LIN {X 65.903,Y 100.037,Z 70.570,A 180.000,B 0.000,C 180.000} C_DIS
LIN {X 65.874,Y 99.882,Z 70.566,A 180.000,B 0.000,C 180.000} C_DIS
LIN {X 65.837,Y 99.729,Z 70.562,A 180.000,B 0.000,C 180.000} C_DIS
LIN {X 65.796,Y 99.577,Z 70.559,A 180.000,B 0.000,C 180.000} C_DIS
LIN {X 65.755,Y 99.425,Z 70.556,A 180.000,B 0.000,C 180.000} C_DIS
LIN {X 65.713,Y 99.273,Z 70.552,A 180.000,B 0.000,C 180.000} C_DIS
LIN {X 65.665,Y 99.123,Z 70.549,A 180.000,B 0.000,C 180.000} C_DIS
LIN {X 65.611,Y 98.975,Z 70.546,A 180.000,B 0.000,C 180.000} C_DIS
LIN {X 65.556,Y 98.827,Z 70.543,A 180.000,B 0.000,C 180.000} C_DIS
LIN {X 65.501,Y 98.679,Z 70.540,A 180.000,B 0.000,C 180.000} C_DIS
LIN {X 65.443,Y 98.533,Z 70.537,A 180.000,B 0.000,C 180.000} C_DIS
LIN {X 65.376,Y 98.391,Z 70.534,A 180.000,B 0.000,C 180.000} C_DIS
LIN {X 65.308,Y 98.248,Z 70.532,A 180.000,B 0.000,C 180.000} C_DIS
LIN {X 65.241,Y 98.106,Z 70.529,A 180.000,B 0.000,C 180.000} C_DIS
LIN {X 65.171,Y 97.965,Z 70.527,A 180.000,B 0.000,C 180.000} C_DIS
LIN {X 65.014,Y 97.692,Z 70.522,A 180.000,B 0.000,C 180.000} C_DIS
LIN {X 64.853,Y 97.421,Z 70.518,A 180.000,B 0.000,C 180.000} C_DIS
LIN {X 64.674,Y 97.162,Z 70.514,A 180.000,B 0.000,C 180.000} C_DIS
LIN {X 64.491,Y 96.906,Z 70.511,A 180.000,B 0.000,C 180.000} C_DIS
LIN {X 64.291,Y 96.662,Z 70.508,A 180.000,B 0.000,C 180.000} C_DIS
LIN {X 64.086,Y 96.423,Z 70.505,A 180.000,B 0.000,C 180.000} C_DIS
LIN {X 63.980,Y 96.307,Z 70.504,A 180.000,B 0.000,C 180.000} C_DIS
LIN {X 63.868,Y 96.196,Z 70.503,A 180.000,B 0.000,C 180.000} C_DIS
LIN {X 63.643,Y 95.976,Z 70.502,A 180.000,B 0.000,C 180.000} C_DIS
LIN {X 63.528,Y 95.868,Z 70.501,A 180.000,B 0.000,C 180.000} C_DIS
LIN {X 63.407,Y 95.766,Z 70.501,A 180.000,B 0.000,C 180.000} C_DIS
LIN {X 63.164,Y 95.567,Z 70.500,A 180.000,B 0.000,C 180.000} C_DIS
LIN {X 62.980,Y 95.424,Z 70.500,A 180.000,B 0.000,C 180.000} C_DIS
; Cutting Move Starts
LIN {X 62.930,Y 95.388,Z 70.500,A 180.000,B 0.000,C 180.000} C_DIS
LIN {X 62.573,Y 95.145,Z 70.500,A 180.000,B 0.000,C 180.000} C_DIS
LIN {X 62.518,Y 95.109,Z 70.500,A 180.000,B 0.000,C 180.000} C_DIS
LIN {X 62.394,Y 95.033,Z 70.500,A 180.000,B 0.000,C 180.000} C_DIS
LIN {X 62.210,Y 94.930,Z 70.500,A 180.000,B 0.000,C 180.000} C_DIS
LIN {X 62.036,Y 94.833,Z 70.500,A 180.000,B 0.000,C 180.000} C_DIS
LIN {X 61.885,Y 94.751,Z 70.500,A 180.000,B 0.000,C 180.000} C_DIS
LIN {X 61.858,Y 94.738,Z 70.500,A 180.000,B 0.000,C 180.000} C_DIS
LIN {X 61.679,Y 94.656,Z 70.500,A 180.000,B 0.000,C 180.000} C_DIS
LIN {X 61.491,Y 94.573,Z 70.500,A 180.000,B 0.000,C 180.000} C_DIS
LIN {X 61.321,Y 94.497,Z 70.500,A 180.000,B 0.000,C 180.000} C_DIS
LIN {X 61.143,Y 94.430,Z 70.500,A 180.000,B 0.000,C 180.000} C_DIS
LIN {X 60.785,Y 94.307,Z 70.500,A 180.000,B 0.000,C 180.000} C_DIS
LIN {X 60.606,Y 94.250,Z 70.500,A 180.000,B 0.000,C 180.000} C_DIS
LIN {X 60.470,Y 94.215,Z 70.500,A 180.000,B 0.000,C 180.000} C_DIS
LIN {X 60.249,Y 94.160,Z 70.500,A 180.000,B 0.000,C 180.000} C_DIS
LIN {X 60.070,Y 94.116,Z 70.500,A 180.000,B 0.000,C 180.000} C_DIS
LIN {X 59.891,Y 94.081,Z 70.500,A 180.000,B 0.000,C 180.000} C_DIS
LIN {X 59.534,Y 94.025,Z 70.500,A 180.000,B 0.000,C 180.000} C_DIS
LIN {X 59.355,Y 93.999,Z 70.500,A 180.000,B 0.000,C 180.000} C_DIS
LIN {X 59.176,Y 93.983,Z 70.500,A 180.000,B 0.000,C 180.000} C_DIS
LIN {X 58.819,Y 93.959,Z 70.500,A 180.000,B 0.000,C 180.000} C_DIS
LIN {X 58.640,Y 93.951,Z 70.500,A 180.000,B 0.000,C 180.000} C_DIS
LIN {X 58.461,Y 93.954,Z 70.500,A 180.000,B 0.000,C 180.000} C_DIS
LIN {X 58.103,Y 93.962,Z 70.500,A 180.000,B 0.000,C 180.000} C_DIS
LIN {X 57.925,Y 93.973,Z 70.500,A 180.000,B 0.000,C 180.000} C_DIS
LIN {X 57.746,Y 93.992,Z 70.500,A 180.000,B 0.000,C 180.000} C_DIS
LIN {X 57.567,Y 94.012,Z 70.500,A 180.000,B 0.000,C 180.000} C_DIS
LIN {X 57.388,Y 94.033,Z 70.500,A 180.000,B 0.000,C 180.000} C_DIS
LIN {X 57.363,Y 94.036,Z 70.500,A 180.000,B 0.000,C 180.000} C_DIS
LIN {X 57.210,Y 94.063,Z 70.500,A 180.000,B 0.000,C 180.000} C_DIS
LIN {X 56.852,Y 94.135,Z 70.500,A 180.000,B 0.000,C 180.000} C_DIS
LIN {X 56.673,Y 94.174,Z 70.500,A 180.000,B 0.000,C 180.000} C_DIS
LIN {X 56.528,Y 94.215,Z 70.500,A 180.000,B 0.000,C 180.000} C_DIS
LIN {X 56.316,Y 94.278,Z 70.500,A 180.000,B 0.000,C 180.000} C_DIS
LIN {X 56.137,Y 94.331,Z 70.500,A 180.000,B 0.000,C 180.000} C_DIS
LIN {X 55.958,Y 94.392,Z 70.500,A 180.000,B 0.000,C 180.000} C_DIS
LIN {X 55.953,Y 94.394,Z 70.500,A 180.000,B 0.000,C 180.000} C_DIS
LIN {X 55.779,Y 94.462,Z 70.500,A 180.000,B 0.000,C 180.000} C_DIS
LIN {X 55.601,Y 94.533,Z 70.500,A 180.000,B 0.000,C 180.000} C_DIS
LIN {X 55.501,Y 94.573,Z 70.500,A 180.000,B 0.000,C 180.000} C_DIS
LIN {X 55.422,Y 94.606,Z 70.500,A 180.000,B 0.000,C 180.000} C_DIS
LIN {X 55.243,Y 94.693,Z 70.500,A 180.000,B 0.000,C 180.000} C_DIS
LIN {X 55.064,Y 94.782,Z 70.500,A 180.000,B 0.000,C 180.000} C_DIS
LIN {X 54.886,Y 94.872,Z 70.500,A 180.000,B 0.000,C 180.000} C_DIS
LIN {X 54.781,Y 94.930,Z 70.500,A 180.000,B 0.000,C 180.000} C_DIS
LIN {X 54.707,Y 94.975,Z 70.500,A 180.000,B 0.000,C 180.000} C_DIS
LIN {X 54.349,Y 95.195,Z 70.500,A 180.000,B 0.000,C 180.000} C_DIS
LIN {X 54.210,Y 95.288,Z 70.500,A 180.000,B 0.000,C 180.000} C_DIS
LIN {X 54.171,Y 95.316,Z 70.500,A 180.000,B 0.000,C 180.000} C_DIS
LIN {X 53.970,Y 95.466,Z 70.500,A 180.000,B 0.000,C 180.000} C_DIS
LIN {X 53.813,Y 95.583,Z 70.500,A 180.000,B 0.000,C 180.000} C_DIS
LIN {X 53.733,Y 95.645,Z 70.500,A 180.000,B 0.000,C 180.000} C_DIS
LIN {X 53.634,Y 95.729,Z 70.500,A 180.000,B 0.000,C 180.000} C_DIS
LIN {X 53.445,Y 95.899,Z 70.500,A 180.000,B 0.000,C 180.000} C_DIS
LIN {X 53.329,Y 96.003,Z 70.500,A 180.000,B 0.000,C 180.000} C_DIS
LIN {X 53.277,Y 96.050,Z 70.500,A 180.000,B 0.000,C 180.000} C_DIS
LIN {X 53.144,Y 96.181,Z 70.500,A 180.000,B 0.000,C 180.000} C_DIS
LIN {X 52.919,Y 96.421,Z 70.500,A 180.000,B 0.000,C 180.000} C_DIS
LIN {X 52.810,Y 96.539,Z 70.500,A 180.000,B 0.000,C 180.000} C_DIS
LIN {X 52.740,Y 96.619,Z 70.500,A 180.000,B 0.000,C 180.000} C_DIS
LIN {X 52.662,Y 96.718,Z 70.500,A 180.000,B 0.000,C 180.000} C_DIS
LIN {X 52.522,Y 96.897,Z 70.500,A 180.000,B 0.000,C 180.000} C_DIS
LIN {X 52.383,Y 97.075,Z 70.500,A 180.000,B 0.000,C 180.000} C_DIS
LIN {X 52.261,Y 97.254,Z 70.500,A 180.000,B 0.000,C 180.000} C_DIS
LIN {X 52.145,Y 97.433,Z 70.500,A 180.000,B 0.000,C 180.000} C_DIS
LIN {X 52.029,Y 97.612,Z 70.500,A 180.000,B 0.000,C 180.000} C_DIS
LIN {X 52.025,Y 97.618,Z 70.500,A 180.000,B 0.000,C 180.000} C_DIS
LIN {X 51.927,Y 97.790,Z 70.500,A 180.000,B 0.000,C 180.000} C_DIS
LIN {X 51.737,Y 98.148,Z 70.500,A 180.000,B 0.000,C 180.000} C_DIS
LIN {X 51.668,Y 98.287,Z 70.500,A 180.000,B 0.000,C 180.000} C_DIS
LIN {X 51.650,Y 98.327,Z 70.500,A 180.000,B 0.000,C 180.000} C_DIS
LIN {X 51.574,Y 98.505,Z 70.500,A 180.000,B 0.000,C 180.000} C_DIS
LIN {X 51.489,Y 98.708,Z 70.500,A 180.000,B 0.000,C 180.000} C_DIS
LIN {X 51.426,Y 98.863,Z 70.500,A 180.000,B 0.000,C 180.000} C_DIS
LIN {X 51.365,Y 99.042,Z 70.500,A 180.000,B 0.000,C 180.000} C_DIS
LIN {X 51.250,Y 99.399,Z 70.500,A 180.000,B 0.000,C 180.000} C_DIS
LIN {X 51.199,Y 99.578,Z 70.500,A 180.000,B 0.000,C 180.000} C_DIS
LIN {X 51.159,Y 99.757,Z 70.500,A 180.000,B 0.000,C 180.000} C_DIS
LIN {X 51.118,Y 99.936,Z 70.500,A 180.000,B 0.000,C 180.000} C_DIS
LIN {X 51.079,Y 100.114,Z 70.500,A 180.000,B 0.000,C 180.000} C_DIS
LIN {X 51.049,Y 100.293,Z 70.500,A 180.000,B 0.000,C 180.000} C_DIS
LIN {X 51.001,Y 100.651,Z 70.500,A 180.000,B 0.000,C 180.000} C_DIS
LIN {X 50.980,Y 100.829,Z 70.500,A 180.000,B 0.000,C 180.000} C_DIS
LIN {X 50.969,Y 101.008,Z 70.500,A 180.000,B 0.000,C 180.000} C_DIS
LIN {X 50.953,Y 101.385,Z 70.500,A 180.000,B 0.000,C 180.000} C_DIS
LIN {X 50.950,Y 101.545,Z 70.500,A 180.000,B 0.000,C 180.000} C_DIS
LIN {X 50.953,Y 101.615,Z 70.500,A 180.000,B 0.000,C 180.000} C_DIS
LIN {X 50.965,Y 101.902,Z 70.500,A 180.000,B 0.000,C 180.000} C_DIS
LIN {X 50.973,Y 102.081,Z 70.500,A 180.000,B 0.000,C 180.000} C_DIS
LIN {X 50.989,Y 102.260,Z 70.500,A 180.000,B 0.000,C 180.000} C_DIS
LIN {X 51.013,Y 102.438,Z 70.500,A 180.000,B 0.000,C 180.000} C_DIS
LIN {X 51.037,Y 102.617,Z 70.500,A 180.000,B 0.000,C 180.000} C_DIS
LIN {X 51.062,Y 102.796,Z 70.500,A 180.000,B 0.000,C 180.000} C_DIS
LIN {X 51.098,Y 102.975,Z 70.500,A 180.000,B 0.000,C 180.000} C_DIS
LIN {X 51.179,Y 103.332,Z 70.500,A 180.000,B 0.000,C 180.000} C_DIS
LIN {X 51.223,Y 103.511,Z 70.500,A 180.000,B 0.000,C 180.000} C_DIS
LIN {X 51.279,Y 103.690,Z 70.500,A 180.000,B 0.000,C 180.000} C_DIS
LIN {X 51.336,Y 103.869,Z 70.500,A 180.000,B 0.000,C 180.000} C_DIS
LIN {X 51.393,Y 104.047,Z 70.500,A 180.000,B 0.000,C 180.000} C_DIS
LIN {X 51.461,Y 104.226,Z 70.500,A 180.000,B 0.000,C 180.000} C_DIS
LIN {X 51.612,Y 104.584,Z 70.500,A 180.000,B 0.000,C 180.000} C_DIS
LIN {X 51.668,Y 104.713,Z 70.500,A 180.000,B 0.000,C 180.000} C_DIS
LIN {X 51.691,Y 104.762,Z 70.500,A 180.000,B 0.000,C 180.000} C_DIS
LIN {X 51.785,Y 104.941,Z 70.500,A 180.000,B 0.000,C 180.000} C_DIS
LIN {X 51.879,Y 105.120,Z 70.500,A 180.000,B 0.000,C 180.000} C_DIS
LIN {X 51.975,Y 105.299,Z 70.500,A 180.000,B 0.000,C 180.000} C_DIS
LIN {X 52.025,Y 105.382,Z 70.500,A 180.000,B 0.000,C 180.000} C_DIS
LIN {X 52.087,Y 105.477,Z 70.500,A 180.000,B 0.000,C 180.000} C_DIS
LIN {X 52.204,Y 105.658,Z 70.500,A 180.000,B 0.000,C 180.000} C_DIS
LIN {X 52.319,Y 105.835,Z 70.500,A 180.000,B 0.000,C 180.000} C_DIS
LIN {X 52.383,Y 105.925,Z 70.500,A 180.000,B 0.000,C 180.000} C_DIS
LIN {X 52.452,Y 106.014,Z 70.500,A 180.000,B 0.000,C 180.000} C_DIS
LIN {X 52.591,Y 106.193,Z 70.500,A 180.000,B 0.000,C 180.000} C_DIS
LIN {X 52.732,Y 106.371,Z 70.500,A 180.000,B 0.000,C 180.000} C_DIS
LIN {X 52.740,Y 106.381,Z 70.500,A 180.000,B 0.000,C 180.000} C_DIS
LIN {X 52.892,Y 106.550,Z 70.500,A 180.000,B 0.000,C 180.000} C_DIS
LIN {X 53.098,Y 106.770,Z 70.500,A 180.000,B 0.000,C 180.000} C_DIS
LIN {X 53.231,Y 106.908,Z 70.500,A 180.000,B 0.000,C 180.000} C_DIS
LIN {X 53.277,Y 106.950,Z 70.500,A 180.000,B 0.000,C 180.000} C_DIS
LIN {X 53.428,Y 107.086,Z 70.500,A 180.000,B 0.000,C 180.000} C_DIS
LIN {X 53.634,Y 107.271,Z 70.500,A 180.000,B 0.000,C 180.000} C_DIS
LIN {X 53.724,Y 107.347,Z 70.500,A 180.000,B 0.000,C 180.000} C_DIS
LIN {X 53.813,Y 107.417,Z 70.500,A 180.000,B 0.000,C 180.000} C_DIS
LIN {X 54.089,Y 107.623,Z 70.500,A 180.000,B 0.000,C 180.000} C_DIS
LIN {X 54.171,Y 107.684,Z 70.500,A 180.000,B 0.000,C 180.000} C_DIS
LIN {X 54.344,Y 107.802,Z 70.500,A 180.000,B 0.000,C 180.000} C_DIS
LIN {X 54.707,Y 108.025,Z 70.500,A 180.000,B 0.000,C 180.000} C_DIS
LIN {X 54.886,Y 108.128,Z 70.500,A 180.000,B 0.000,C 180.000} C_DIS
LIN {X 54.947,Y 108.159,Z 70.500,A 180.000,B 0.000,C 180.000} C_DIS
LIN {X 55.304,Y 108.338,Z 70.500,A 180.000,B 0.000,C 180.000} C_DIS
LIN {X 55.422,Y 108.394,Z 70.500,A 180.000,B 0.000,C 180.000} C_DIS
LIN {X 55.601,Y 108.467,Z 70.500,A 180.000,B 0.000,C 180.000} C_DIS
LIN {X 55.779,Y 108.538,Z 70.500,A 180.000,B 0.000,C 180.000} C_DIS
LIN {X 55.958,Y 108.608,Z 70.500,A 180.000,B 0.000,C 180.000} C_DIS
LIN {X 56.137,Y 108.669,Z 70.500,A 180.000,B 0.000,C 180.000} C_DIS
LIN {X 56.225,Y 108.695,Z 70.500,A 180.000,B 0.000,C 180.000} C_DIS
LIN {X 56.495,Y 108.775,Z 70.500,A 180.000,B 0.000,C 180.000} C_DIS
LIN {X 56.673,Y 108.826,Z 70.500,A 180.000,B 0.000,C 180.000} C_DIS
LIN {X 56.852,Y 108.865,Z 70.500,A 180.000,B 0.000,C 180.000} C_DIS
LIN {X 57.210,Y 108.937,Z 70.500,A 180.000,B 0.000,C 180.000} C_DIS
LIN {X 57.388,Y 108.967,Z 70.500,A 180.000,B 0.000,C 180.000} C_DIS
LIN {X 57.567,Y 108.988,Z 70.500,A 180.000,B 0.000,C 180.000} C_DIS
LIN {X 57.746,Y 109.008,Z 70.500,A 180.000,B 0.000,C 180.000} C_DIS
LIN {X 57.925,Y 109.027,Z 70.500,A 180.000,B 0.000,C 180.000} C_DIS
LIN {X 58.103,Y 109.038,Z 70.500,A 180.000,B 0.000,C 180.000} C_DIS
LIN {X 58.461,Y 109.046,Z 70.500,A 180.000,B 0.000,C 180.000} C_DIS
LIN {X 58.640,Y 109.049,Z 70.500,A 180.000,B 0.000,C 180.000} C_DIS
LIN {X 58.819,Y 109.041,Z 70.500,A 180.000,B 0.000,C 180.000} C_DIS
LIN {X 59.176,Y 109.017,Z 70.500,A 180.000,B 0.000,C 180.000} C_DIS
LIN {X 59.355,Y 109.001,Z 70.500,A 180.000,B 0.000,C 180.000} C_DIS
LIN {X 59.534,Y 108.975,Z 70.500,A 180.000,B 0.000,C 180.000} C_DIS
LIN {X 59.891,Y 108.919,Z 70.500,A 180.000,B 0.000,C 180.000} C_DIS
LIN {X 60.070,Y 108.884,Z 70.500,A 180.000,B 0.000,C 180.000} C_DIS
LIN {X 60.111,Y 108.874,Z 70.500,A 180.000,B 0.000,C 180.000} C_DIS
LIN {X 60.427,Y 108.796,Z 70.500,A 180.000,B 0.000,C 180.000} C_DIS
LIN {X 60.606,Y 108.750,Z 70.500,A 180.000,B 0.000,C 180.000} C_DIS
LIN {X 60.778,Y 108.695,Z 70.500,A 180.000,B 0.000,C 180.000} C_DIS
LIN {X 61.143,Y 108.570,Z 70.500,A 180.000,B 0.000,C 180.000} C_DIS
LIN {X 61.287,Y 108.517,Z 70.500,A 180.000,B 0.000,C 180.000} C_DIS
LIN {X 61.321,Y 108.503,Z 70.500,A 180.000,B 0.000,C 180.000} C_DIS
LIN {X 61.500,Y 108.424,Z 70.500,A 180.000,B 0.000,C 180.000} C_DIS
LIN {X 61.692,Y 108.338,Z 70.500,A 180.000,B 0.000,C 180.000} C_DIS
LIN {X 61.858,Y 108.262,Z 70.500,A 180.000,B 0.000,C 180.000} C_DIS
LIN {X 62.036,Y 108.167,Z 70.500,A 180.000,B 0.000,C 180.000} C_DIS
LIN {X 62.371,Y 107.980,Z 70.500,A 180.000,B 0.000,C 180.000} C_DIS
LIN {X 62.394,Y 107.967,Z 70.500,A 180.000,B 0.000,C 180.000} C_DIS
LIN {X 62.573,Y 107.855,Z 70.500,A 180.000,B 0.000,C 180.000} C_DIS
LIN {X 62.930,Y 107.612,Z 70.500,A 180.000,B 0.000,C 180.000} C_DIS
LIN {X 63.020,Y 107.548,Z 70.500,A 180.000,B 0.000,C 180.000} C_DIS
LIN {X 63.109,Y 107.478,Z 70.500,A 180.000,B 0.000,C 180.000} C_DIS
LIN {X 63.369,Y 107.265,Z 70.500,A 180.000,B 0.000,C 180.000} C_DIS
LIN {X 63.467,Y 107.185,Z 70.500,A 180.000,B 0.000,C 180.000} C_DIS
LIN {X 63.578,Y 107.086,Z 70.500,A 180.000,B 0.000,C 180.000} C_DIS
LIN {X 63.645,Y 107.021,Z 70.500,A 180.000,B 0.000,C 180.000} C_DIS
LIN {X 63.824,Y 106.847,Z 70.500,A 180.000,B 0.000,C 180.000} C_DIS
LIN {X 63.944,Y 106.729,Z 70.500,A 180.000,B 0.000,C 180.000} C_DIS
LIN {X 64.003,Y 106.669,Z 70.500,A 180.000,B 0.000,C 180.000} C_DIS
LIN {X 64.109,Y 106.550,Z 70.500,A 180.000,B 0.000,C 180.000} C_DIS
LIN {X 64.360,Y 106.256,Z 70.500,A 180.000,B 0.000,C 180.000} C_DIS
LIN {X 64.414,Y 106.193,Z 70.500,A 180.000,B 0.000,C 180.000} C_DIS
LIN {X 64.539,Y 106.026,Z 70.500,A 180.000,B 0.000,C 180.000} C_DIS
LIN {X 64.718,Y 105.776,Z 70.500,A 180.000,B 0.000,C 180.000} C_DIS
LIN {X 64.802,Y 105.656,Z 70.500,A 180.000,B 0.000,C 180.000} C_DIS
LIN {X 64.897,Y 105.507,Z 70.500,A 180.000,B 0.000,C 180.000} C_DIS
LIN {X 65.075,Y 105.203,Z 70.500,A 180.000,B 0.000,C 180.000} C_DIS
LIN {X 65.124,Y 105.120,Z 70.500,A 180.000,B 0.000,C 180.000} C_DIS
LIN {X 65.219,Y 104.941,Z 70.500,A 180.000,B 0.000,C 180.000} C_DIS
LIN {X 65.254,Y 104.866,Z 70.500,A 180.000,B 0.000,C 180.000} C_DIS
LIN {X 65.388,Y 104.584,Z 70.500,A 180.000,B 0.000,C 180.000} C_DIS
LIN {X 65.433,Y 104.488,Z 70.500,A 180.000,B 0.000,C 180.000} C_DIS
LIN {X 65.469,Y 104.405,Z 70.500,A 180.000,B 0.000,C 180.000} C_DIS
LIN {X 65.536,Y 104.226,Z 70.500,A 180.000,B 0.000,C 180.000} C_DIS
LIN {X 65.612,Y 104.022,Z 70.500,A 180.000,B 0.000,C 180.000} C_DIS
LIN {X 65.668,Y 103.869,Z 70.500,A 180.000,B 0.000,C 180.000} C_DIS
LIN {X 65.724,Y 103.690,Z 70.500,A 180.000,B 0.000,C 180.000} C_DIS
LIN {X 65.821,Y 103.332,Z 70.500,A 180.000,B 0.000,C 180.000} C_DIS
LIN {X 65.867,Y 103.153,Z 70.500,A 180.000,B 0.000,C 180.000} C_DIS
LIN {X 65.901,Y 102.975,Z 70.500,A 180.000,B 0.000,C 180.000} C_DIS
LIN {X 65.965,Y 102.617,Z 70.500,A 180.000,B 0.000,C 180.000} C_DIS
LIN {X 65.969,Y 102.592,Z 70.500,A 180.000,B 0.000,C 180.000} C_DIS
LIN {X 65.991,Y 102.438,Z 70.500,A 180.000,B 0.000,C 180.000} C_DIS
LIN {X 66.007,Y 102.260,Z 70.500,A 180.000,B 0.000,C 180.000} C_DIS
LIN {X 66.023,Y 102.081,Z 70.500,A 180.000,B 0.000,C 180.000} C_DIS
LIN {X 66.039,Y 101.902,Z 70.500,A 180.000,B 0.000,C 180.000} C_DIS
LIN {X 66.045,Y 101.723,Z 70.500,A 180.000,B 0.000,C 180.000} C_DIS
LIN {X 66.045,Y 101.366,Z 70.500,A 180.000,B 0.000,C 180.000} C_DIS
LIN {X 66.043,Y 101.187,Z 70.500,A 180.000,B 0.000,C 180.000} C_DIS
LIN {X 66.031,Y 101.008,Z 70.500,A 180.000,B 0.000,C 180.000} C_DIS
LIN {X 65.999,Y 100.651,Z 70.500,A 180.000,B 0.000,C 180.000} C_DIS
LIN {X 65.980,Y 100.472,Z 70.500,A 180.000,B 0.000,C 180.000} C_DIS
LIN {X 65.969,Y 100.408,Z 70.500,A 180.000,B 0.000,C 180.000} C_DIS
LIN {X 65.949,Y 100.293,Z 70.500,A 180.000,B 0.000,C 180.000} C_DIS
LIN {X 65.917,Y 100.114,Z 70.500,A 180.000,B 0.000,C 180.000} C_DIS
LIN {X 65.885,Y 99.936,Z 70.500,A 180.000,B 0.000,C 180.000} C_DIS
LIN {X 65.845,Y 99.757,Z 70.500,A 180.000,B 0.000,C 180.000} C_DIS
LIN {X 65.796,Y 99.578,Z 70.500,A 180.000,B 0.000,C 180.000} C_DIS
LIN {X 65.748,Y 99.399,Z 70.500,A 180.000,B 0.000,C 180.000} C_DIS
LIN {X 65.698,Y 99.221,Z 70.500,A 180.000,B 0.000,C 180.000} C_DIS
LIN {X 65.635,Y 99.042,Z 70.500,A 180.000,B 0.000,C 180.000} C_DIS
LIN {X 65.503,Y 98.684,Z 70.500,A 180.000,B 0.000,C 180.000} C_DIS
LIN {X 65.433,Y 98.512,Z 70.500,A 180.000,B 0.000,C 180.000} C_DIS
LIN {X 65.430,Y 98.505,Z 70.500,A 180.000,B 0.000,C 180.000} C_DIS
LIN {X 65.346,Y 98.327,Z 70.500,A 180.000,B 0.000,C 180.000} C_DIS
LIN {X 65.254,Y 98.134,Z 70.500,A 180.000,B 0.000,C 180.000} C_DIS
LIN {X 65.174,Y 97.969,Z 70.500,A 180.000,B 0.000,C 180.000} C_DIS
LIN {X 65.075,Y 97.797,Z 70.500,A 180.000,B 0.000,C 180.000} C_DIS
LIN {X 64.897,Y 97.493,Z 70.500,A 180.000,B 0.000,C 180.000} C_DIS
LIN {X 64.861,Y 97.433,Z 70.500,A 180.000,B 0.000,C 180.000} C_DIS
LIN {X 64.739,Y 97.254,Z 70.500,A 180.000,B 0.000,C 180.000} C_DIS
LIN {X 64.539,Y 96.974,Z 70.500,A 180.000,B 0.000,C 180.000} C_DIS
LIN {X 64.484,Y 96.897,Z 70.500,A 180.000,B 0.000,C 180.000} C_DIS
LIN {X 64.360,Y 96.744,Z 70.500,A 180.000,B 0.000,C 180.000} C_DIS
LIN {X 64.182,Y 96.535,Z 70.500,A 180.000,B 0.000,C 180.000} C_DIS
LIN {X 64.030,Y 96.360,Z 70.500,A 180.000,B 0.000,C 180.000} C_DIS
LIN {X 64.003,Y 96.331,Z 70.500,A 180.000,B 0.000,C 180.000} C_DIS
LIN {X 63.853,Y 96.181,Z 70.500,A 180.000,B 0.000,C 180.000} C_DIS
LIN {X 63.645,Y 95.979,Z 70.500,A 180.000,B 0.000,C 180.000} C_DIS
LIN {X 63.477,Y 95.824,Z 70.500,A 180.000,B 0.000,C 180.000} C_DIS
LIN {X 63.467,Y 95.815,Z 70.500,A 180.000,B 0.000,C 180.000} C_DIS
LIN {X 63.288,Y 95.669,Z 70.500,A 180.000,B 0.000,C 180.000} C_DIS
LIN {X 63.109,Y 95.522,Z 70.500,A 180.000,B 0.000,C 180.000} C_DIS
LIN {X 63.038,Y 95.466,Z 70.500,A 180.000,B 0.000,C 180.000} C_DIS
LIN {X 62.980,Y 95.424,Z 70.500,A 180.000,B 0.000,C 180.000} C_DIS
; Link Move Starts
LIN {X 62.722,Y 95.246,Z 70.499,A 180.000,B 0.000,C 180.000} C_DIS
LIN {X 62.461,Y 95.072,Z 70.496,A 180.000,B 0.000,C 180.000} C_DIS
LIN {X 62.188,Y 94.918,Z 70.492,A 180.000,B 0.000,C 180.000} C_DIS
LIN {X 62.051,Y 94.841,Z 70.489,A 180.000,B 0.000,C 180.000} C_DIS
LIN {X 61.914,Y 94.766,Z 70.486,A 180.000,B 0.000,C 180.000} C_DIS
LIN {X 61.772,Y 94.698,Z 70.482,A 180.000,B 0.000,C 180.000} C_DIS
LIN {X 61.629,Y 94.634,Z 70.479,A 180.000,B 0.000,C 180.000} C_DIS
LIN {X 61.486,Y 94.570,Z 70.475,A 180.000,B 0.000,C 180.000} C_DIS
LIN {X 61.343,Y 94.506,Z 70.470,A 180.000,B 0.000,C 180.000} C_DIS
LIN {X 61.197,Y 94.449,Z 70.465,A 180.000,B 0.000,C 180.000} C_DIS
LIN {X 61.049,Y 94.398,Z 70.460,A 180.000,B 0.000,C 180.000} C_DIS
LIN {X 60.975,Y 94.372,Z 70.458,A 180.000,B 0.000,C 180.000} C_DIS
LIN {X 60.900,Y 94.347,Z 70.455,A 180.000,B 0.000,C 180.000} C_DIS
LIN {X 60.826,Y 94.321,Z 70.453,A 180.000,B 0.000,C 180.000} C_DIS
LIN {X 60.752,Y 94.296,Z 70.450,A 180.000,B 0.000,C 180.000} C_DIS
LIN {X 60.678,Y 94.271,Z 70.447,A 180.000,B 0.000,C 180.000} C_DIS
LIN {X 60.603,Y 94.249,Z 70.444,A 180.000,B 0.000,C 180.000} C_DIS
LIN {X 60.527,Y 94.229,Z 70.442,A 180.000,B 0.000,C 180.000} C_DIS
LIN {X 60.451,Y 94.210,Z 70.439,A 180.000,B 0.000,C 180.000} C_DIS
LIN {X 60.375,Y 94.191,Z 70.436,A 180.000,B 0.000,C 180.000} C_DIS
LIN {X 60.298,Y 94.172,Z 70.433,A 180.000,B 0.000,C 180.000} C_DIS
LIN {X 60.222,Y 94.153,Z 70.431,A 180.000,B 0.000,C 180.000} C_DIS
LIN {X 60.146,Y 94.135,Z 70.428,A 180.000,B 0.000,C 180.000} C_DIS
LIN {X 60.070,Y 94.116,Z 70.425,A 180.000,B 0.000,C 180.000} C_DIS
LIN {X 59.994,Y 94.099,Z 70.422,A 180.000,B 0.000,C 180.000} C_DIS
LIN {X 59.916,Y 94.085,Z 70.420,A 180.000,B 0.000,C 180.000} C_DIS
LIN {X 59.839,Y 94.073,Z 70.417,A 180.000,B 0.000,C 180.000} C_DIS
LIN {X 59.762,Y 94.060,Z 70.414,A 180.000,B 0.000,C 180.000} C_DIS
LIN {X 59.684,Y 94.048,Z 70.411,A 180.000,B 0.000,C 180.000} C_DIS
LIN {X 59.607,Y 94.036,Z 70.409,A 180.000,B 0.000,C 180.000} C_DIS
LIN {X 59.529,Y 94.024,Z 70.406,A 180.000,B 0.000,C 180.000} C_DIS
LIN {X 59.452,Y 94.012,Z 70.403,A 180.000,B 0.000,C 180.000} C_DIS
LIN {X 59.374,Y 94.001,Z 70.401,A 180.000,B 0.000,C 180.000} C_DIS
LIN {X 59.296,Y 93.992,Z 70.398,A 180.000,B 0.000,C 180.000} C_DIS
LIN {X 59.218,Y 93.986,Z 70.395,A 180.000,B 0.000,C 180.000} C_DIS
LIN {X 59.062,Y 93.976,Z 70.390,A 180.000,B 0.000,C 180.000} C_DIS
LIN {X 58.827,Y 93.960,Z 70.381,A 180.000,B 0.000,C 180.000} C_DIS
LIN {X 58.749,Y 93.955,Z 70.379,A 180.000,B 0.000,C 180.000} C_DIS
LIN {X 58.670,Y 93.952,Z 70.376,A 180.000,B 0.000,C 180.000} C_DIS
LIN {X 58.592,Y 93.951,Z 70.373,A 180.000,B 0.000,C 180.000} C_DIS
LIN {X 58.514,Y 93.953,Z 70.370,A 180.000,B 0.000,C 180.000} C_DIS
LIN {X 58.122,Y 93.961,Z 70.357,A 180.000,B 0.000,C 180.000} C_DIS
LIN {X 58.043,Y 93.964,Z 70.354,A 180.000,B 0.000,C 180.000} C_DIS
LIN {X 57.965,Y 93.969,Z 70.351,A 180.000,B 0.000,C 180.000} C_DIS
LIN {X 57.887,Y 93.977,Z 70.348,A 180.000,B 0.000,C 180.000} C_DIS
LIN {X 57.731,Y 93.994,Z 70.343,A 180.000,B 0.000,C 180.000} C_DIS
LIN {X 57.653,Y 94.003,Z 70.340,A 180.000,B 0.000,C 180.000} C_DIS
LIN {X 57.575,Y 94.011,Z 70.338,A 180.000,B 0.000,C 180.000} C_DIS
LIN {X 57.497,Y 94.020,Z 70.335,A 180.000,B 0.000,C 180.000} C_DIS
LIN {X 57.420,Y 94.029,Z 70.332,A 180.000,B 0.000,C 180.000} C_DIS
LIN {X 57.342,Y 94.039,Z 70.329,A 180.000,B 0.000,C 180.000} C_DIS
LIN {X 57.265,Y 94.052,Z 70.327,A 180.000,B 0.000,C 180.000} C_DIS
LIN {X 57.188,Y 94.068,Z 70.324,A 180.000,B 0.000,C 180.000} C_DIS
LIN {X 57.111,Y 94.083,Z 70.321,A 180.000,B 0.000,C 180.000} C_DIS
LIN {X 57.034,Y 94.099,Z 70.318,A 180.000,B 0.000,C 180.000} C_DIS
LIN {X 56.957,Y 94.114,Z 70.316,A 180.000,B 0.000,C 180.000} C_DIS
LIN {X 56.880,Y 94.130,Z 70.313,A 180.000,B 0.000,C 180.000} C_DIS
LIN {X 56.803,Y 94.145,Z 70.310,A 180.000,B 0.000,C 180.000} C_DIS
LIN {X 56.727,Y 94.162,Z 70.307,A 180.000,B 0.000,C 180.000} C_DIS
LIN {X 56.651,Y 94.180,Z 70.305,A 180.000,B 0.000,C 180.000} C_DIS
LIN {X 56.575,Y 94.201,Z 70.302,A 180.000,B 0.000,C 180.000} C_DIS
LIN {X 56.500,Y 94.223,Z 70.299,A 180.000,B 0.000,C 180.000} C_DIS
LIN {X 56.425,Y 94.246,Z 70.297,A 180.000,B 0.000,C 180.000} C_DIS
LIN {X 56.349,Y 94.268,Z 70.294,A 180.000,B 0.000,C 180.000} C_DIS
LIN {X 56.274,Y 94.290,Z 70.291,A 180.000,B 0.000,C 180.000} C_DIS
LIN {X 56.199,Y 94.312,Z 70.288,A 180.000,B 0.000,C 180.000} C_DIS
LIN {X 56.124,Y 94.335,Z 70.286,A 180.000,B 0.000,C 180.000} C_DIS
LIN {X 55.976,Y 94.385,Z 70.281,A 180.000,B 0.000,C 180.000} C_DIS
LIN {X 55.830,Y 94.442,Z 70.276,A 180.000,B 0.000,C 180.000} C_DIS
LIN {X 55.684,Y 94.500,Z 70.272,A 180.000,B 0.000,C 180.000} C_DIS
LIN {X 55.538,Y 94.558,Z 70.268,A 180.000,B 0.000,C 180.000} C_DIS
LIN {X 55.394,Y 94.619,Z 70.264,A 180.000,B 0.000,C 180.000} C_DIS
LIN {X 55.253,Y 94.688,Z 70.260,A 180.000,B 0.000,C 180.000} C_DIS
LIN {X 55.113,Y 94.758,Z 70.257,A 180.000,B 0.000,C 180.000} C_DIS
LIN {X 54.972,Y 94.828,Z 70.255,A 180.000,B 0.000,C 180.000} C_DIS
LIN {X 54.833,Y 94.900,Z 70.252,A 180.000,B 0.000,C 180.000} C_DIS
LIN {X 54.698,Y 94.980,Z 70.250,A 180.000,B 0.000,C 180.000} C_DIS
LIN {X 54.431,Y 95.145,Z 70.247,A 180.000,B 0.000,C 180.000} C_DIS
LIN {X 54.177,Y 95.312,Z 70.247,A 180.000,B 0.000,C 180.000} C_DIS
; Cutting Move Starts
LIN {X 54.171,Y 95.316,Z 70.247,A 180.000,B 0.000,C 180.000} C_DIS
LIN {X 53.970,Y 95.466,Z 70.247,A 180.000,B 0.000,C 180.000} C_DIS
LIN {X 53.813,Y 95.583,Z 70.247,A 180.000,B 0.000,C 180.000} C_DIS
LIN {X 53.733,Y 95.645,Z 70.247,A 180.000,B 0.000,C 180.000} C_DIS
LIN {X 53.634,Y 95.729,Z 70.247,A 180.000,B 0.000,C 180.000} C_DIS
LIN {X 53.329,Y 96.003,Z 70.247,A 180.000,B 0.000,C 180.000} C_DIS
LIN {X 53.277,Y 96.050,Z 70.247,A 180.000,B 0.000,C 180.000} C_DIS
LIN {X 53.144,Y 96.181,Z 70.247,A 180.000,B 0.000,C 180.000} C_DIS
LIN {X 52.919,Y 96.421,Z 70.247,A 180.000,B 0.000,C 180.000} C_DIS
LIN {X 52.810,Y 96.539,Z 70.247,A 180.000,B 0.000,C 180.000} C_DIS
LIN {X 52.740,Y 96.619,Z 70.247,A 180.000,B 0.000,C 180.000} C_DIS
LIN {X 52.662,Y 96.718,Z 70.247,A 180.000,B 0.000,C 180.000} C_DIS
LIN {X 52.522,Y 96.897,Z 70.247,A 180.000,B 0.000,C 180.000} C_DIS
LIN {X 52.383,Y 97.075,Z 70.247,A 180.000,B 0.000,C 180.000} C_DIS
LIN {X 52.261,Y 97.254,Z 70.247,A 180.000,B 0.000,C 180.000} C_DIS
LIN {X 52.145,Y 97.433,Z 70.247,A 180.000,B 0.000,C 180.000} C_DIS
LIN {X 52.029,Y 97.612,Z 70.247,A 180.000,B 0.000,C 180.000} C_DIS
LIN {X 52.025,Y 97.618,Z 70.247,A 180.000,B 0.000,C 180.000} C_DIS
LIN {X 51.927,Y 97.790,Z 70.247,A 180.000,B 0.000,C 180.000} C_DIS
LIN {X 51.737,Y 98.148,Z 70.247,A 180.000,B 0.000,C 180.000} C_DIS
LIN {X 51.668,Y 98.287,Z 70.247,A 180.000,B 0.000,C 180.000} C_DIS
LIN {X 51.650,Y 98.327,Z 70.247,A 180.000,B 0.000,C 180.000} C_DIS
LIN {X 51.574,Y 98.505,Z 70.247,A 180.000,B 0.000,C 180.000} C_DIS
LIN {X 51.489,Y 98.708,Z 70.247,A 180.000,B 0.000,C 180.000} C_DIS
LIN {X 51.426,Y 98.863,Z 70.247,A 180.000,B 0.000,C 180.000} C_DIS
LIN {X 51.365,Y 99.042,Z 70.247,A 180.000,B 0.000,C 180.000} C_DIS
LIN {X 51.250,Y 99.399,Z 70.247,A 180.000,B 0.000,C 180.000} C_DIS
LIN {X 51.199,Y 99.578,Z 70.247,A 180.000,B 0.000,C 180.000} C_DIS
LIN {X 51.159,Y 99.757,Z 70.247,A 180.000,B 0.000,C 180.000} C_DIS
LIN {X 51.118,Y 99.936,Z 70.247,A 180.000,B 0.000,C 180.000} C_DIS
LIN {X 51.079,Y 100.114,Z 70.247,A 180.000,B 0.000,C 180.000} C_DIS
LIN {X 51.049,Y 100.293,Z 70.247,A 180.000,B 0.000,C 180.000} C_DIS
LIN {X 51.001,Y 100.651,Z 70.247,A 180.000,B 0.000,C 180.000} C_DIS
LIN {X 50.980,Y 100.829,Z 70.247,A 180.000,B 0.000,C 180.000} C_DIS
LIN {X 50.969,Y 101.008,Z 70.247,A 180.000,B 0.000,C 180.000} C_DIS
LIN {X 50.953,Y 101.385,Z 70.247,A 180.000,B 0.000,C 180.000} C_DIS
LIN {X 50.950,Y 101.545,Z 70.247,A 180.000,B 0.000,C 180.000} C_DIS
LIN {X 50.953,Y 101.615,Z 70.247,A 180.000,B 0.000,C 180.000} C_DIS
LIN {X 50.965,Y 101.902,Z 70.247,A 180.000,B 0.000,C 180.000} C_DIS
LIN {X 50.973,Y 102.081,Z 70.247,A 180.000,B 0.000,C 180.000} C_DIS
LIN {X 50.989,Y 102.260,Z 70.247,A 180.000,B 0.000,C 180.000} C_DIS
LIN {X 51.013,Y 102.438,Z 70.247,A 180.000,B 0.000,C 180.000} C_DIS
LIN {X 51.037,Y 102.617,Z 70.247,A 180.000,B 0.000,C 180.000} C_DIS
LIN {X 51.062,Y 102.796,Z 70.247,A 180.000,B 0.000,C 180.000} C_DIS
LIN {X 51.098,Y 102.975,Z 70.247,A 180.000,B 0.000,C 180.000} C_DIS
LIN {X 51.179,Y 103.332,Z 70.247,A 180.000,B 0.000,C 180.000} C_DIS
LIN {X 51.223,Y 103.511,Z 70.247,A 180.000,B 0.000,C 180.000} C_DIS
LIN {X 51.279,Y 103.690,Z 70.247,A 180.000,B 0.000,C 180.000} C_DIS
LIN {X 51.336,Y 103.869,Z 70.247,A 180.000,B 0.000,C 180.000} C_DIS
LIN {X 51.393,Y 104.047,Z 70.247,A 180.000,B 0.000,C 180.000} C_DIS
LIN {X 51.461,Y 104.226,Z 70.247,A 180.000,B 0.000,C 180.000} C_DIS
LIN {X 51.612,Y 104.584,Z 70.247,A 180.000,B 0.000,C 180.000} C_DIS
LIN {X 51.668,Y 104.713,Z 70.247,A 180.000,B 0.000,C 180.000} C_DIS
LIN {X 51.691,Y 104.762,Z 70.247,A 180.000,B 0.000,C 180.000} C_DIS
LIN {X 51.785,Y 104.941,Z 70.247,A 180.000,B 0.000,C 180.000} C_DIS
LIN {X 51.879,Y 105.120,Z 70.247,A 180.000,B 0.000,C 180.000} C_DIS
LIN {X 51.975,Y 105.299,Z 70.247,A 180.000,B 0.000,C 180.000} C_DIS
LIN {X 52.025,Y 105.382,Z 70.247,A 180.000,B 0.000,C 180.000} C_DIS
LIN {X 52.087,Y 105.477,Z 70.247,A 180.000,B 0.000,C 180.000} C_DIS
LIN {X 52.204,Y 105.658,Z 70.247,A 180.000,B 0.000,C 180.000} C_DIS
LIN {X 52.319,Y 105.835,Z 70.247,A 180.000,B 0.000,C 180.000} C_DIS
LIN {X 52.383,Y 105.925,Z 70.247,A 180.000,B 0.000,C 180.000} C_DIS
LIN {X 52.452,Y 106.014,Z 70.247,A 180.000,B 0.000,C 180.000} C_DIS
LIN {X 52.591,Y 106.193,Z 70.247,A 180.000,B 0.000,C 180.000} C_DIS
LIN {X 52.732,Y 106.371,Z 70.247,A 180.000,B 0.000,C 180.000} C_DIS
LIN {X 52.740,Y 106.381,Z 70.247,A 180.000,B 0.000,C 180.000} C_DIS
LIN {X 52.892,Y 106.550,Z 70.247,A 180.000,B 0.000,C 180.000} C_DIS
LIN {X 53.098,Y 106.770,Z 70.247,A 180.000,B 0.000,C 180.000} C_DIS
LIN {X 53.231,Y 106.908,Z 70.247,A 180.000,B 0.000,C 180.000} C_DIS
LIN {X 53.277,Y 106.950,Z 70.247,A 180.000,B 0.000,C 180.000} C_DIS
LIN {X 53.428,Y 107.086,Z 70.247,A 180.000,B 0.000,C 180.000} C_DIS
LIN {X 53.634,Y 107.271,Z 70.247,A 180.000,B 0.000,C 180.000} C_DIS
LIN {X 53.724,Y 107.347,Z 70.247,A 180.000,B 0.000,C 180.000} C_DIS
LIN {X 53.813,Y 107.417,Z 70.247,A 180.000,B 0.000,C 180.000} C_DIS
LIN {X 54.089,Y 107.623,Z 70.247,A 180.000,B 0.000,C 180.000} C_DIS
LIN {X 54.171,Y 107.684,Z 70.247,A 180.000,B 0.000,C 180.000} C_DIS
LIN {X 54.344,Y 107.802,Z 70.247,A 180.000,B 0.000,C 180.000} C_DIS
LIN {X 54.707,Y 108.025,Z 70.247,A 180.000,B 0.000,C 180.000} C_DIS
LIN {X 54.886,Y 108.128,Z 70.247,A 180.000,B 0.000,C 180.000} C_DIS
LIN {X 54.947,Y 108.159,Z 70.247,A 180.000,B 0.000,C 180.000} C_DIS
LIN {X 55.304,Y 108.338,Z 70.247,A 180.000,B 0.000,C 180.000} C_DIS
LIN {X 55.422,Y 108.394,Z 70.247,A 180.000,B 0.000,C 180.000} C_DIS
LIN {X 55.601,Y 108.467,Z 70.247,A 180.000,B 0.000,C 180.000} C_DIS
LIN {X 55.779,Y 108.538,Z 70.247,A 180.000,B 0.000,C 180.000} C_DIS
LIN {X 55.958,Y 108.608,Z 70.247,A 180.000,B 0.000,C 180.000} C_DIS
LIN {X 56.137,Y 108.669,Z 70.247,A 180.000,B 0.000,C 180.000} C_DIS
LIN {X 56.225,Y 108.695,Z 70.247,A 180.000,B 0.000,C 180.000} C_DIS
LIN {X 56.495,Y 108.775,Z 70.247,A 180.000,B 0.000,C 180.000} C_DIS
LIN {X 56.673,Y 108.826,Z 70.247,A 180.000,B 0.000,C 180.000} C_DIS
LIN {X 56.852,Y 108.865,Z 70.247,A 180.000,B 0.000,C 180.000} C_DIS
LIN {X 57.210,Y 108.937,Z 70.247,A 180.000,B 0.000,C 180.000} C_DIS
LIN {X 57.388,Y 108.967,Z 70.247,A 180.000,B 0.000,C 180.000} C_DIS
LIN {X 57.567,Y 108.988,Z 70.247,A 180.000,B 0.000,C 180.000} C_DIS
LIN {X 57.746,Y 109.008,Z 70.247,A 180.000,B 0.000,C 180.000} C_DIS
LIN {X 57.925,Y 109.027,Z 70.247,A 180.000,B 0.000,C 180.000} C_DIS
LIN {X 58.103,Y 109.038,Z 70.247,A 180.000,B 0.000,C 180.000} C_DIS
LIN {X 58.461,Y 109.046,Z 70.247,A 180.000,B 0.000,C 180.000} C_DIS
LIN {X 58.640,Y 109.049,Z 70.247,A 180.000,B 0.000,C 180.000} C_DIS
LIN {X 58.819,Y 109.041,Z 70.247,A 180.000,B 0.000,C 180.000} C_DIS
LIN {X 59.176,Y 109.017,Z 70.247,A 180.000,B 0.000,C 180.000} C_DIS
LIN {X 59.355,Y 109.001,Z 70.247,A 180.000,B 0.000,C 180.000} C_DIS
LIN {X 59.534,Y 108.975,Z 70.247,A 180.000,B 0.000,C 180.000} C_DIS
LIN {X 59.891,Y 108.919,Z 70.247,A 180.000,B 0.000,C 180.000} C_DIS
LIN {X 60.070,Y 108.884,Z 70.247,A 180.000,B 0.000,C 180.000} C_DIS
LIN {X 60.111,Y 108.874,Z 70.247,A 180.000,B 0.000,C 180.000} C_DIS
LIN {X 60.427,Y 108.796,Z 70.247,A 180.000,B 0.000,C 180.000} C_DIS
LIN {X 60.606,Y 108.750,Z 70.247,A 180.000,B 0.000,C 180.000} C_DIS
LIN {X 60.778,Y 108.695,Z 70.247,A 180.000,B 0.000,C 180.000} C_DIS
LIN {X 61.143,Y 108.570,Z 70.247,A 180.000,B 0.000,C 180.000} C_DIS
LIN {X 61.287,Y 108.517,Z 70.247,A 180.000,B 0.000,C 180.000} C_DIS
LIN {X 61.321,Y 108.503,Z 70.247,A 180.000,B 0.000,C 180.000} C_DIS
LIN {X 61.500,Y 108.424,Z 70.247,A 180.000,B 0.000,C 180.000} C_DIS
LIN {X 61.692,Y 108.338,Z 70.247,A 180.000,B 0.000,C 180.000} C_DIS
LIN {X 61.858,Y 108.262,Z 70.247,A 180.000,B 0.000,C 180.000} C_DIS
LIN {X 62.036,Y 108.167,Z 70.247,A 180.000,B 0.000,C 180.000} C_DIS
LIN {X 62.371,Y 107.980,Z 70.247,A 180.000,B 0.000,C 180.000} C_DIS
LIN {X 62.394,Y 107.967,Z 70.247,A 180.000,B 0.000,C 180.000} C_DIS
LIN {X 62.573,Y 107.855,Z 70.247,A 180.000,B 0.000,C 180.000} C_DIS
LIN {X 62.930,Y 107.612,Z 70.247,A 180.000,B 0.000,C 180.000} C_DIS
LIN {X 63.020,Y 107.548,Z 70.247,A 180.000,B 0.000,C 180.000} C_DIS
LIN {X 63.109,Y 107.478,Z 70.247,A 180.000,B 0.000,C 180.000} C_DIS
LIN {X 63.369,Y 107.265,Z 70.247,A 180.000,B 0.000,C 180.000} C_DIS
LIN {X 63.467,Y 107.185,Z 70.247,A 180.000,B 0.000,C 180.000} C_DIS
LIN {X 63.578,Y 107.086,Z 70.247,A 180.000,B 0.000,C 180.000} C_DIS
LIN {X 63.645,Y 107.021,Z 70.247,A 180.000,B 0.000,C 180.000} C_DIS
LIN {X 63.824,Y 106.847,Z 70.247,A 180.000,B 0.000,C 180.000} C_DIS
LIN {X 63.944,Y 106.729,Z 70.247,A 180.000,B 0.000,C 180.000} C_DIS
LIN {X 64.003,Y 106.669,Z 70.247,A 180.000,B 0.000,C 180.000} C_DIS
LIN {X 64.109,Y 106.550,Z 70.247,A 180.000,B 0.000,C 180.000} C_DIS
LIN {X 64.360,Y 106.256,Z 70.247,A 180.000,B 0.000,C 180.000} C_DIS
LIN {X 64.414,Y 106.193,Z 70.247,A 180.000,B 0.000,C 180.000} C_DIS
LIN {X 64.539,Y 106.026,Z 70.247,A 180.000,B 0.000,C 180.000} C_DIS
LIN {X 64.718,Y 105.776,Z 70.247,A 180.000,B 0.000,C 180.000} C_DIS
LIN {X 64.802,Y 105.656,Z 70.247,A 180.000,B 0.000,C 180.000} C_DIS
LIN {X 64.897,Y 105.507,Z 70.247,A 180.000,B 0.000,C 180.000} C_DIS
LIN {X 65.075,Y 105.203,Z 70.247,A 180.000,B 0.000,C 180.000} C_DIS
LIN {X 65.124,Y 105.120,Z 70.247,A 180.000,B 0.000,C 180.000} C_DIS
LIN {X 65.219,Y 104.941,Z 70.247,A 180.000,B 0.000,C 180.000} C_DIS
LIN {X 65.254,Y 104.866,Z 70.247,A 180.000,B 0.000,C 180.000} C_DIS
LIN {X 65.388,Y 104.584,Z 70.247,A 180.000,B 0.000,C 180.000} C_DIS
LIN {X 65.433,Y 104.488,Z 70.247,A 180.000,B 0.000,C 180.000} C_DIS
LIN {X 65.469,Y 104.405,Z 70.247,A 180.000,B 0.000,C 180.000} C_DIS
LIN {X 65.536,Y 104.226,Z 70.247,A 180.000,B 0.000,C 180.000} C_DIS
LIN {X 65.612,Y 104.022,Z 70.247,A 180.000,B 0.000,C 180.000} C_DIS
LIN {X 65.668,Y 103.869,Z 70.247,A 180.000,B 0.000,C 180.000} C_DIS
LIN {X 65.724,Y 103.690,Z 70.247,A 180.000,B 0.000,C 180.000} C_DIS
LIN {X 65.821,Y 103.332,Z 70.247,A 180.000,B 0.000,C 180.000} C_DIS
LIN {X 65.867,Y 103.153,Z 70.247,A 180.000,B 0.000,C 180.000} C_DIS
LIN {X 65.901,Y 102.975,Z 70.247,A 180.000,B 0.000,C 180.000} C_DIS
LIN {X 65.965,Y 102.617,Z 70.247,A 180.000,B 0.000,C 180.000} C_DIS
LIN {X 65.969,Y 102.592,Z 70.247,A 180.000,B 0.000,C 180.000} C_DIS
LIN {X 65.991,Y 102.438,Z 70.247,A 180.000,B 0.000,C 180.000} C_DIS
LIN {X 66.007,Y 102.260,Z 70.247,A 180.000,B 0.000,C 180.000} C_DIS
LIN {X 66.023,Y 102.081,Z 70.247,A 180.000,B 0.000,C 180.000} C_DIS
LIN {X 66.039,Y 101.902,Z 70.247,A 180.000,B 0.000,C 180.000} C_DIS
LIN {X 66.045,Y 101.723,Z 70.247,A 180.000,B 0.000,C 180.000} C_DIS
LIN {X 66.045,Y 101.366,Z 70.247,A 180.000,B 0.000,C 180.000} C_DIS
LIN {X 66.043,Y 101.187,Z 70.247,A 180.000,B 0.000,C 180.000} C_DIS
LIN {X 66.031,Y 101.008,Z 70.247,A 180.000,B 0.000,C 180.000} C_DIS
LIN {X 65.999,Y 100.651,Z 70.247,A 180.000,B 0.000,C 180.000} C_DIS
LIN {X 65.980,Y 100.472,Z 70.247,A 180.000,B 0.000,C 180.000} C_DIS
LIN {X 65.969,Y 100.408,Z 70.247,A 180.000,B 0.000,C 180.000} C_DIS
LIN {X 65.949,Y 100.293,Z 70.247,A 180.000,B 0.000,C 180.000} C_DIS
LIN {X 65.917,Y 100.114,Z 70.247,A 180.000,B 0.000,C 180.000} C_DIS
LIN {X 65.885,Y 99.936,Z 70.247,A 180.000,B 0.000,C 180.000} C_DIS
LIN {X 65.845,Y 99.757,Z 70.247,A 180.000,B 0.000,C 180.000} C_DIS
LIN {X 65.796,Y 99.578,Z 70.247,A 180.000,B 0.000,C 180.000} C_DIS
LIN {X 65.748,Y 99.399,Z 70.247,A 180.000,B 0.000,C 180.000} C_DIS
LIN {X 65.698,Y 99.221,Z 70.247,A 180.000,B 0.000,C 180.000} C_DIS
LIN {X 65.635,Y 99.042,Z 70.247,A 180.000,B 0.000,C 180.000} C_DIS
LIN {X 65.503,Y 98.684,Z 70.247,A 180.000,B 0.000,C 180.000} C_DIS
LIN {X 65.433,Y 98.512,Z 70.247,A 180.000,B 0.000,C 180.000} C_DIS
LIN {X 65.430,Y 98.505,Z 70.247,A 180.000,B 0.000,C 180.000} C_DIS
LIN {X 65.346,Y 98.327,Z 70.247,A 180.000,B 0.000,C 180.000} C_DIS
LIN {X 65.254,Y 98.134,Z 70.247,A 180.000,B 0.000,C 180.000} C_DIS
LIN {X 65.174,Y 97.969,Z 70.247,A 180.000,B 0.000,C 180.000} C_DIS
LIN {X 65.075,Y 97.797,Z 70.247,A 180.000,B 0.000,C 180.000} C_DIS
LIN {X 64.897,Y 97.493,Z 70.247,A 180.000,B 0.000,C 180.000} C_DIS
LIN {X 64.861,Y 97.433,Z 70.247,A 180.000,B 0.000,C 180.000} C_DIS
LIN {X 64.739,Y 97.254,Z 70.247,A 180.000,B 0.000,C 180.000} C_DIS
LIN {X 64.539,Y 96.974,Z 70.247,A 180.000,B 0.000,C 180.000} C_DIS
LIN {X 64.484,Y 96.897,Z 70.247,A 180.000,B 0.000,C 180.000} C_DIS
LIN {X 64.360,Y 96.744,Z 70.247,A 180.000,B 0.000,C 180.000} C_DIS
LIN {X 64.182,Y 96.535,Z 70.247,A 180.000,B 0.000,C 180.000} C_DIS
LIN {X 64.030,Y 96.360,Z 70.247,A 180.000,B 0.000,C 180.000} C_DIS
LIN {X 64.003,Y 96.331,Z 70.247,A 180.000,B 0.000,C 180.000} C_DIS
LIN {X 63.853,Y 96.181,Z 70.247,A 180.000,B 0.000,C 180.000} C_DIS
LIN {X 63.645,Y 95.979,Z 70.247,A 180.000,B 0.000,C 180.000} C_DIS
LIN {X 63.477,Y 95.824,Z 70.247,A 180.000,B 0.000,C 180.000} C_DIS
LIN {X 63.467,Y 95.815,Z 70.247,A 180.000,B 0.000,C 180.000} C_DIS
LIN {X 63.288,Y 95.669,Z 70.247,A 180.000,B 0.000,C 180.000} C_DIS
LIN {X 63.109,Y 95.522,Z 70.247,A 180.000,B 0.000,C 180.000} C_DIS
LIN {X 63.038,Y 95.466,Z 70.247,A 180.000,B 0.000,C 180.000} C_DIS
LIN {X 62.980,Y 95.424,Z 70.247,A 180.000,B 0.000,C 180.000} C_DIS
LIN {X 62.930,Y 95.388,Z 70.247,A 180.000,B 0.000,C 180.000} C_DIS
LIN {X 62.573,Y 95.145,Z 70.247,A 180.000,B 0.000,C 180.000} C_DIS
LIN {X 62.518,Y 95.109,Z 70.247,A 180.000,B 0.000,C 180.000} C_DIS
LIN {X 62.394,Y 95.033,Z 70.247,A 180.000,B 0.000,C 180.000} C_DIS
LIN {X 62.210,Y 94.930,Z 70.247,A 180.000,B 0.000,C 180.000} C_DIS
LIN {X 62.036,Y 94.833,Z 70.247,A 180.000,B 0.000,C 180.000} C_DIS
LIN {X 61.885,Y 94.751,Z 70.247,A 180.000,B 0.000,C 180.000} C_DIS
LIN {X 61.858,Y 94.738,Z 70.247,A 180.000,B 0.000,C 180.000} C_DIS
LIN {X 61.679,Y 94.656,Z 70.247,A 180.000,B 0.000,C 180.000} C_DIS
LIN {X 61.491,Y 94.573,Z 70.247,A 180.000,B 0.000,C 180.000} C_DIS
LIN {X 61.321,Y 94.497,Z 70.247,A 180.000,B 0.000,C 180.000} C_DIS
LIN {X 61.143,Y 94.430,Z 70.247,A 180.000,B 0.000,C 180.000} C_DIS
LIN {X 60.785,Y 94.307,Z 70.247,A 180.000,B 0.000,C 180.000} C_DIS
LIN {X 60.606,Y 94.250,Z 70.247,A 180.000,B 0.000,C 180.000} C_DIS
LIN {X 60.470,Y 94.215,Z 70.247,A 180.000,B 0.000,C 180.000} C_DIS
LIN {X 60.249,Y 94.160,Z 70.247,A 180.000,B 0.000,C 180.000} C_DIS
LIN {X 60.070,Y 94.116,Z 70.247,A 180.000,B 0.000,C 180.000} C_DIS
LIN {X 59.891,Y 94.081,Z 70.247,A 180.000,B 0.000,C 180.000} C_DIS
LIN {X 59.534,Y 94.025,Z 70.247,A 180.000,B 0.000,C 180.000} C_DIS
LIN {X 59.355,Y 93.999,Z 70.247,A 180.000,B 0.000,C 180.000} C_DIS
LIN {X 59.176,Y 93.983,Z 70.247,A 180.000,B 0.000,C 180.000} C_DIS
LIN {X 58.819,Y 93.959,Z 70.247,A 180.000,B 0.000,C 180.000} C_DIS
LIN {X 58.640,Y 93.951,Z 70.247,A 180.000,B 0.000,C 180.000} C_DIS
LIN {X 58.461,Y 93.954,Z 70.247,A 180.000,B 0.000,C 180.000} C_DIS
LIN {X 58.103,Y 93.962,Z 70.247,A 180.000,B 0.000,C 180.000} C_DIS
LIN {X 57.925,Y 93.973,Z 70.247,A 180.000,B 0.000,C 180.000} C_DIS
LIN {X 57.746,Y 93.992,Z 70.247,A 180.000,B 0.000,C 180.000} C_DIS
LIN {X 57.567,Y 94.012,Z 70.247,A 180.000,B 0.000,C 180.000} C_DIS
LIN {X 57.388,Y 94.033,Z 70.247,A 180.000,B 0.000,C 180.000} C_DIS
LIN {X 57.363,Y 94.036,Z 70.247,A 180.000,B 0.000,C 180.000} C_DIS
LIN {X 57.210,Y 94.063,Z 70.247,A 180.000,B 0.000,C 180.000} C_DIS
LIN {X 56.852,Y 94.135,Z 70.247,A 180.000,B 0.000,C 180.000} C_DIS
LIN {X 56.673,Y 94.174,Z 70.247,A 180.000,B 0.000,C 180.000} C_DIS
LIN {X 56.528,Y 94.215,Z 70.247,A 180.000,B 0.000,C 180.000} C_DIS
LIN {X 56.316,Y 94.278,Z 70.247,A 180.000,B 0.000,C 180.000} C_DIS
LIN {X 56.137,Y 94.331,Z 70.247,A 180.000,B 0.000,C 180.000} C_DIS
LIN {X 55.958,Y 94.392,Z 70.247,A 180.000,B 0.000,C 180.000} C_DIS
LIN {X 55.953,Y 94.394,Z 70.247,A 180.000,B 0.000,C 180.000} C_DIS
LIN {X 55.779,Y 94.462,Z 70.247,A 180.000,B 0.000,C 180.000} C_DIS
LIN {X 55.601,Y 94.533,Z 70.247,A 180.000,B 0.000,C 180.000} C_DIS
LIN {X 55.501,Y 94.573,Z 70.247,A 180.000,B 0.000,C 180.000} C_DIS
LIN {X 55.422,Y 94.606,Z 70.247,A 180.000,B 0.000,C 180.000} C_DIS
LIN {X 55.243,Y 94.693,Z 70.247,A 180.000,B 0.000,C 180.000} C_DIS
LIN {X 55.064,Y 94.782,Z 70.247,A 180.000,B 0.000,C 180.000} C_DIS
LIN {X 54.886,Y 94.872,Z 70.247,A 180.000,B 0.000,C 180.000} C_DIS
LIN {X 54.781,Y 94.930,Z 70.247,A 180.000,B 0.000,C 180.000} C_DIS
LIN {X 54.707,Y 94.975,Z 70.247,A 180.000,B 0.000,C 180.000} C_DIS
LIN {X 54.349,Y 95.195,Z 70.247,A 180.000,B 0.000,C 180.000} C_DIS
LIN {X 54.210,Y 95.288,Z 70.247,A 180.000,B 0.000,C 180.000} C_DIS
LIN {X 54.177,Y 95.312,Z 70.247,A 180.000,B 0.000,C 180.000} C_DIS
; Link Move Starts
LIN {X 53.933,Y 95.494,Z 70.246,A 180.000,B 0.000,C 180.000} C_DIS
LIN {X 53.691,Y 95.680,Z 70.243,A 180.000,B 0.000,C 180.000} C_DIS
LIN {X 53.463,Y 95.883,Z 70.239,A 180.000,B 0.000,C 180.000} C_DIS
LIN {X 53.349,Y 95.985,Z 70.236,A 180.000,B 0.000,C 180.000} C_DIS
LIN {X 53.236,Y 96.087,Z 70.233,A 180.000,B 0.000,C 180.000} C_DIS
LIN {X 53.130,Y 96.196,Z 70.230,A 180.000,B 0.000,C 180.000} C_DIS
LIN {X 53.025,Y 96.308,Z 70.226,A 180.000,B 0.000,C 180.000} C_DIS
LIN {X 52.921,Y 96.419,Z 70.222,A 180.000,B 0.000,C 180.000} C_DIS
LIN {X 52.817,Y 96.531,Z 70.217,A 180.000,B 0.000,C 180.000} C_DIS
LIN {X 52.718,Y 96.647,Z 70.213,A 180.000,B 0.000,C 180.000} C_DIS
LIN {X 52.623,Y 96.767,Z 70.208,A 180.000,B 0.000,C 180.000} C_DIS
LIN {X 52.576,Y 96.827,Z 70.206,A 180.000,B 0.000,C 180.000} C_DIS
LIN {X 52.529,Y 96.887,Z 70.203,A 180.000,B 0.000,C 180.000} C_DIS
LIN {X 52.482,Y 96.947,Z 70.200,A 180.000,B 0.000,C 180.000} C_DIS
LIN {X 52.435,Y 97.007,Z 70.198,A 180.000,B 0.000,C 180.000} C_DIS
LIN {X 52.389,Y 97.067,Z 70.195,A 180.000,B 0.000,C 180.000} C_DIS
LIN {X 52.344,Y 97.129,Z 70.192,A 180.000,B 0.000,C 180.000} C_DIS
LIN {X 52.301,Y 97.192,Z 70.190,A 180.000,B 0.000,C 180.000} C_DIS
LIN {X 52.259,Y 97.256,Z 70.187,A 180.000,B 0.000,C 180.000} C_DIS
LIN {X 52.218,Y 97.320,Z 70.184,A 180.000,B 0.000,C 180.000} C_DIS
LIN {X 52.176,Y 97.384,Z 70.182,A 180.000,B 0.000,C 180.000} C_DIS
LIN {X 52.135,Y 97.448,Z 70.179,A 180.000,B 0.000,C 180.000} C_DIS
LIN {X 52.093,Y 97.512,Z 70.176,A 180.000,B 0.000,C 180.000} C_DIS
LIN {X 52.052,Y 97.576,Z 70.174,A 180.000,B 0.000,C 180.000} C_DIS
LIN {X 52.011,Y 97.641,Z 70.171,A 180.000,B 0.000,C 180.000} C_DIS
LIN {X 51.972,Y 97.707,Z 70.168,A 180.000,B 0.000,C 180.000} C_DIS
LIN {X 51.936,Y 97.773,Z 70.166,A 180.000,B 0.000,C 180.000} C_DIS
LIN {X 51.900,Y 97.841,Z 70.163,A 180.000,B 0.000,C 180.000} C_DIS
LIN {X 51.864,Y 97.908,Z 70.160,A 180.000,B 0.000,C 180.000} C_DIS
LIN {X 51.829,Y 97.976,Z 70.158,A 180.000,B 0.000,C 180.000} C_DIS
LIN {X 51.793,Y 98.043,Z 70.155,A 180.000,B 0.000,C 180.000} C_DIS
LIN {X 51.757,Y 98.111,Z 70.152,A 180.000,B 0.000,C 180.000} C_DIS
LIN {X 51.722,Y 98.178,Z 70.150,A 180.000,B 0.000,C 180.000} C_DIS
LIN {X 51.687,Y 98.246,Z 70.147,A 180.000,B 0.000,C 180.000} C_DIS
LIN {X 51.655,Y 98.315,Z 70.144,A 180.000,B 0.000,C 180.000} C_DIS
LIN {X 51.625,Y 98.385,Z 70.142,A 180.000,B 0.000,C 180.000} C_DIS
LIN {X 51.566,Y 98.526,Z 70.136,A 180.000,B 0.000,C 180.000} C_DIS
LIN {X 51.506,Y 98.667,Z 70.131,A 180.000,B 0.000,C 180.000} C_DIS
LIN {X 51.477,Y 98.737,Z 70.128,A 180.000,B 0.000,C 180.000} C_DIS
LIN {X 51.447,Y 98.807,Z 70.126,A 180.000,B 0.000,C 180.000} C_DIS
LIN {X 51.420,Y 98.878,Z 70.123,A 180.000,B 0.000,C 180.000} C_DIS
LIN {X 51.394,Y 98.950,Z 70.120,A 180.000,B 0.000,C 180.000} C_DIS
LIN {X 51.371,Y 99.023,Z 70.118,A 180.000,B 0.000,C 180.000} C_DIS
LIN {X 51.254,Y 99.386,Z 70.104,A 180.000,B 0.000,C 180.000} C_DIS
LIN {X 51.232,Y 99.459,Z 70.102,A 180.000,B 0.000,C 180.000} C_DIS
LIN {X 51.211,Y 99.533,Z 70.099,A 180.000,B 0.000,C 180.000} C_DIS
LIN {X 51.192,Y 99.607,Z 70.096,A 180.000,B 0.000,C 180.000} C_DIS
LIN {X 51.176,Y 99.681,Z 70.094,A 180.000,B 0.000,C 180.000} C_DIS
LIN {X 51.159,Y 99.755,Z 70.091,A 180.000,B 0.000,C 180.000} C_DIS
LIN {X 51.142,Y 99.830,Z 70.088,A 180.000,B 0.000,C 180.000} C_DIS
LIN {X 51.125,Y 99.904,Z 70.086,A 180.000,B 0.000,C 180.000} C_DIS
LIN {X 51.109,Y 99.979,Z 70.083,A 180.000,B 0.000,C 180.000} C_DIS
LIN {X 51.092,Y 100.053,Z 70.081,A 180.000,B 0.000,C 180.000} C_DIS
LIN {X 51.076,Y 100.128,Z 70.078,A 180.000,B 0.000,C 180.000} C_DIS
LIN {X 51.062,Y 100.203,Z 70.075,A 180.000,B 0.000,C 180.000} C_DIS
LIN {X 51.051,Y 100.278,Z 70.072,A 180.000,B 0.000,C 180.000} C_DIS
LIN {X 51.041,Y 100.354,Z 70.070,A 180.000,B 0.000,C 180.000} C_DIS
LIN {X 51.031,Y 100.430,Z 70.067,A 180.000,B 0.000,C 180.000} C_DIS
LIN {X 51.021,Y 100.505,Z 70.064,A 180.000,B 0.000,C 180.000} C_DIS
LIN {X 51.011,Y 100.581,Z 70.062,A 180.000,B 0.000,C 180.000} C_DIS
LIN {X 51.001,Y 100.656,Z 70.059,A 180.000,B 0.000,C 180.000} C_DIS
LIN {X 50.991,Y 100.732,Z 70.056,A 180.000,B 0.000,C 180.000} C_DIS
LIN {X 50.982,Y 100.808,Z 70.054,A 180.000,B 0.000,C 180.000} C_DIS
LIN {X 50.976,Y 100.884,Z 70.051,A 180.000,B 0.000,C 180.000} C_DIS
LIN {X 50.971,Y 100.960,Z 70.049,A 180.000,B 0.000,C 180.000} C_DIS
LIN {X 50.968,Y 101.036,Z 70.046,A 180.000,B 0.000,C 180.000} C_DIS
LIN {X 50.965,Y 101.112,Z 70.043,A 180.000,B 0.000,C 180.000} C_DIS
LIN {X 50.961,Y 101.189,Z 70.041,A 180.000,B 0.000,C 180.000} C_DIS
LIN {X 50.958,Y 101.265,Z 70.038,A 180.000,B 0.000,C 180.000} C_DIS
LIN {X 50.951,Y 101.417,Z 70.033,A 180.000,B 0.000,C 180.000} C_DIS
LIN {X 50.951,Y 101.570,Z 70.029,A 180.000,B 0.000,C 180.000} C_DIS
LIN {X 50.957,Y 101.722,Z 70.025,A 180.000,B 0.000,C 180.000} C_DIS
LIN {X 50.964,Y 101.875,Z 70.021,A 180.000,B 0.000,C 180.000} C_DIS
LIN {X 50.971,Y 102.027,Z 70.017,A 180.000,B 0.000,C 180.000} C_DIS
LIN {X 50.981,Y 102.180,Z 70.013,A 180.000,B 0.000,C 180.000} C_DIS
LIN {X 50.999,Y 102.331,Z 70.010,A 180.000,B 0.000,C 180.000} C_DIS
LIN {X 51.019,Y 102.482,Z 70.008,A 180.000,B 0.000,C 180.000} C_DIS
LIN {X 51.060,Y 102.785,Z 70.003,A 180.000,B 0.000,C 180.000} C_DIS
LIN {X 51.123,Y 103.083,Z 70.001,A 180.000,B 0.000,C 180.000} C_DIS
LIN {X 51.188,Y 103.372,Z 70.000,A 180.000,B 0.000,C 180.000} C_DIS
; Cutting Move Starts
LIN {X 51.223,Y 103.511,Z 70.000,A 180.000,B 0.000,C 180.000} C_DIS
LIN {X 51.279,Y 103.690,Z 70.000,A 180.000,B 0.000,C 180.000} C_DIS
LIN {X 51.336,Y 103.869,Z 70.000,A 180.000,B 0.000,C 180.000} C_DIS
LIN {X 51.393,Y 104.047,Z 70.000,A 180.000,B 0.000,C 180.000} C_DIS
LIN {X 51.461,Y 104.226,Z 70.000,A 180.000,B 0.000,C 180.000} C_DIS
LIN {X 51.612,Y 104.584,Z 70.000,A 180.000,B 0.000,C 180.000} C_DIS
LIN {X 51.668,Y 104.713,Z 70.000,A 180.000,B 0.000,C 180.000} C_DIS
LIN {X 51.691,Y 104.762,Z 70.000,A 180.000,B 0.000,C 180.000} C_DIS
LIN {X 51.785,Y 104.941,Z 70.000,A 180.000,B 0.000,C 180.000} C_DIS
LIN {X 51.879,Y 105.120,Z 70.000,A 180.000,B 0.000,C 180.000} C_DIS
LIN {X 51.975,Y 105.299,Z 70.000,A 180.000,B 0.000,C 180.000} C_DIS
LIN {X 52.025,Y 105.382,Z 70.000,A 180.000,B 0.000,C 180.000} C_DIS
LIN {X 52.087,Y 105.477,Z 70.000,A 180.000,B 0.000,C 180.000} C_DIS
LIN {X 52.204,Y 105.658,Z 70.000,A 180.000,B 0.000,C 180.000} C_DIS
LIN {X 52.319,Y 105.835,Z 70.000,A 180.000,B 0.000,C 180.000} C_DIS
LIN {X 52.383,Y 105.925,Z 70.000,A 180.000,B 0.000,C 180.000} C_DIS
LIN {X 52.452,Y 106.014,Z 70.000,A 180.000,B 0.000,C 180.000} C_DIS
LIN {X 52.591,Y 106.193,Z 70.000,A 180.000,B 0.000,C 180.000} C_DIS
LIN {X 52.732,Y 106.371,Z 70.000,A 180.000,B 0.000,C 180.000} C_DIS
LIN {X 52.740,Y 106.381,Z 70.000,A 180.000,B 0.000,C 180.000} C_DIS
LIN {X 52.892,Y 106.550,Z 70.000,A 180.000,B 0.000,C 180.000} C_DIS
LIN {X 53.098,Y 106.770,Z 70.000,A 180.000,B 0.000,C 180.000} C_DIS
LIN {X 53.231,Y 106.908,Z 70.000,A 180.000,B 0.000,C 180.000} C_DIS
LIN {X 53.277,Y 106.950,Z 70.000,A 180.000,B 0.000,C 180.000} C_DIS
LIN {X 53.428,Y 107.086,Z 70.000,A 180.000,B 0.000,C 180.000} C_DIS
LIN {X 53.634,Y 107.271,Z 70.000,A 180.000,B 0.000,C 180.000} C_DIS
LIN {X 53.724,Y 107.347,Z 70.000,A 180.000,B 0.000,C 180.000} C_DIS
LIN {X 53.813,Y 107.417,Z 70.000,A 180.000,B 0.000,C 180.000} C_DIS
LIN {X 54.089,Y 107.623,Z 70.000,A 180.000,B 0.000,C 180.000} C_DIS
LIN {X 54.171,Y 107.684,Z 70.000,A 180.000,B 0.000,C 180.000} C_DIS
LIN {X 54.344,Y 107.802,Z 70.000,A 180.000,B 0.000,C 180.000} C_DIS
LIN {X 54.707,Y 108.025,Z 70.000,A 180.000,B 0.000,C 180.000} C_DIS
LIN {X 54.886,Y 108.128,Z 70.000,A 180.000,B 0.000,C 180.000} C_DIS
LIN {X 54.947,Y 108.159,Z 70.000,A 180.000,B 0.000,C 180.000} C_DIS
LIN {X 55.304,Y 108.338,Z 70.000,A 180.000,B 0.000,C 180.000} C_DIS
LIN {X 55.422,Y 108.394,Z 70.000,A 180.000,B 0.000,C 180.000} C_DIS
LIN {X 55.601,Y 108.467,Z 70.000,A 180.000,B 0.000,C 180.000} C_DIS
LIN {X 55.779,Y 108.538,Z 70.000,A 180.000,B 0.000,C 180.000} C_DIS
LIN {X 55.958,Y 108.608,Z 70.000,A 180.000,B 0.000,C 180.000} C_DIS
LIN {X 56.137,Y 108.669,Z 70.000,A 180.000,B 0.000,C 180.000} C_DIS
LIN {X 56.225,Y 108.695,Z 70.000,A 180.000,B 0.000,C 180.000} C_DIS
LIN {X 56.495,Y 108.775,Z 70.000,A 180.000,B 0.000,C 180.000} C_DIS
LIN {X 56.673,Y 108.826,Z 70.000,A 180.000,B 0.000,C 180.000} C_DIS
LIN {X 56.852,Y 108.865,Z 70.000,A 180.000,B 0.000,C 180.000} C_DIS
LIN {X 57.210,Y 108.937,Z 70.000,A 180.000,B 0.000,C 180.000} C_DIS
LIN {X 57.388,Y 108.967,Z 70.000,A 180.000,B 0.000,C 180.000} C_DIS
LIN {X 57.567,Y 108.988,Z 70.000,A 180.000,B 0.000,C 180.000} C_DIS
LIN {X 57.746,Y 109.008,Z 70.000,A 180.000,B 0.000,C 180.000} C_DIS
LIN {X 57.925,Y 109.027,Z 70.000,A 180.000,B 0.000,C 180.000} C_DIS
LIN {X 58.103,Y 109.038,Z 70.000,A 180.000,B 0.000,C 180.000} C_DIS
LIN {X 58.461,Y 109.046,Z 70.000,A 180.000,B 0.000,C 180.000} C_DIS
LIN {X 58.640,Y 109.049,Z 70.000,A 180.000,B 0.000,C 180.000} C_DIS
LIN {X 58.819,Y 109.041,Z 70.000,A 180.000,B 0.000,C 180.000} C_DIS
LIN {X 59.176,Y 109.017,Z 70.000,A 180.000,B 0.000,C 180.000} C_DIS
LIN {X 59.355,Y 109.001,Z 70.000,A 180.000,B 0.000,C 180.000} C_DIS
LIN {X 59.534,Y 108.975,Z 70.000,A 180.000,B 0.000,C 180.000} C_DIS
LIN {X 59.891,Y 108.919,Z 70.000,A 180.000,B 0.000,C 180.000} C_DIS
LIN {X 60.070,Y 108.884,Z 70.000,A 180.000,B 0.000,C 180.000} C_DIS
LIN {X 60.111,Y 108.874,Z 70.000,A 180.000,B 0.000,C 180.000} C_DIS
LIN {X 60.427,Y 108.796,Z 70.000,A 180.000,B 0.000,C 180.000} C_DIS
LIN {X 60.606,Y 108.750,Z 70.000,A 180.000,B 0.000,C 180.000} C_DIS
LIN {X 60.778,Y 108.695,Z 70.000,A 180.000,B 0.000,C 180.000} C_DIS
LIN {X 61.143,Y 108.570,Z 70.000,A 180.000,B 0.000,C 180.000} C_DIS
LIN {X 61.287,Y 108.517,Z 70.000,A 180.000,B 0.000,C 180.000} C_DIS
LIN {X 61.321,Y 108.503,Z 70.000,A 180.000,B 0.000,C 180.000} C_DIS
LIN {X 61.500,Y 108.424,Z 70.000,A 180.000,B 0.000,C 180.000} C_DIS
LIN {X 61.692,Y 108.338,Z 70.000,A 180.000,B 0.000,C 180.000} C_DIS
LIN {X 61.858,Y 108.262,Z 70.000,A 180.000,B 0.000,C 180.000} C_DIS
LIN {X 62.036,Y 108.167,Z 70.000,A 180.000,B 0.000,C 180.000} C_DIS
LIN {X 62.371,Y 107.980,Z 70.000,A 180.000,B 0.000,C 180.000} C_DIS
LIN {X 62.394,Y 107.967,Z 70.000,A 180.000,B 0.000,C 180.000} C_DIS
LIN {X 62.573,Y 107.855,Z 70.000,A 180.000,B 0.000,C 180.000} C_DIS
LIN {X 62.930,Y 107.612,Z 70.000,A 180.000,B 0.000,C 180.000} C_DIS
LIN {X 63.020,Y 107.548,Z 70.000,A 180.000,B 0.000,C 180.000} C_DIS
LIN {X 63.109,Y 107.478,Z 70.000,A 180.000,B 0.000,C 180.000} C_DIS
LIN {X 63.369,Y 107.265,Z 70.000,A 180.000,B 0.000,C 180.000} C_DIS
LIN {X 63.467,Y 107.185,Z 70.000,A 180.000,B 0.000,C 180.000} C_DIS
LIN {X 63.578,Y 107.086,Z 70.000,A 180.000,B 0.000,C 180.000} C_DIS
LIN {X 63.645,Y 107.021,Z 70.000,A 180.000,B 0.000,C 180.000} C_DIS
LIN {X 63.824,Y 106.847,Z 70.000,A 180.000,B 0.000,C 180.000} C_DIS
LIN {X 63.944,Y 106.729,Z 70.000,A 180.000,B 0.000,C 180.000} C_DIS
LIN {X 64.003,Y 106.669,Z 70.000,A 180.000,B 0.000,C 180.000} C_DIS
LIN {X 64.109,Y 106.550,Z 70.000,A 180.000,B 0.000,C 180.000} C_DIS
LIN {X 64.360,Y 106.256,Z 70.000,A 180.000,B 0.000,C 180.000} C_DIS
LIN {X 64.414,Y 106.193,Z 70.000,A 180.000,B 0.000,C 180.000} C_DIS
LIN {X 64.539,Y 106.026,Z 70.000,A 180.000,B 0.000,C 180.000} C_DIS
LIN {X 64.718,Y 105.776,Z 70.000,A 180.000,B 0.000,C 180.000} C_DIS
LIN {X 64.802,Y 105.656,Z 70.000,A 180.000,B 0.000,C 180.000} C_DIS
LIN {X 64.897,Y 105.507,Z 70.000,A 180.000,B 0.000,C 180.000} C_DIS
LIN {X 65.075,Y 105.203,Z 70.000,A 180.000,B 0.000,C 180.000} C_DIS
LIN {X 65.124,Y 105.120,Z 70.000,A 180.000,B 0.000,C 180.000} C_DIS
LIN {X 65.219,Y 104.941,Z 70.000,A 180.000,B 0.000,C 180.000} C_DIS
LIN {X 65.254,Y 104.866,Z 70.000,A 180.000,B 0.000,C 180.000} C_DIS
LIN {X 65.388,Y 104.584,Z 70.000,A 180.000,B 0.000,C 180.000} C_DIS
LIN {X 65.433,Y 104.488,Z 70.000,A 180.000,B 0.000,C 180.000} C_DIS
LIN {X 65.469,Y 104.405,Z 70.000,A 180.000,B 0.000,C 180.000} C_DIS
LIN {X 65.536,Y 104.226,Z 70.000,A 180.000,B 0.000,C 180.000} C_DIS
LIN {X 65.612,Y 104.022,Z 70.000,A 180.000,B 0.000,C 180.000} C_DIS
LIN {X 65.668,Y 103.869,Z 70.000,A 180.000,B 0.000,C 180.000} C_DIS
LIN {X 65.724,Y 103.690,Z 70.000,A 180.000,B 0.000,C 180.000} C_DIS
LIN {X 65.821,Y 103.332,Z 70.000,A 180.000,B 0.000,C 180.000} C_DIS
LIN {X 65.867,Y 103.153,Z 70.000,A 180.000,B 0.000,C 180.000} C_DIS
LIN {X 65.901,Y 102.975,Z 70.000,A 180.000,B 0.000,C 180.000} C_DIS
LIN {X 65.965,Y 102.617,Z 70.000,A 180.000,B 0.000,C 180.000} C_DIS
LIN {X 65.969,Y 102.592,Z 70.000,A 180.000,B 0.000,C 180.000} C_DIS
LIN {X 65.991,Y 102.438,Z 70.000,A 180.000,B 0.000,C 180.000} C_DIS
LIN {X 66.007,Y 102.260,Z 70.000,A 180.000,B 0.000,C 180.000} C_DIS
LIN {X 66.023,Y 102.081,Z 70.000,A 180.000,B 0.000,C 180.000} C_DIS
LIN {X 66.039,Y 101.902,Z 70.000,A 180.000,B 0.000,C 180.000} C_DIS
LIN {X 66.045,Y 101.723,Z 70.000,A 180.000,B 0.000,C 180.000} C_DIS
LIN {X 66.045,Y 101.366,Z 70.000,A 180.000,B 0.000,C 180.000} C_DIS
LIN {X 66.043,Y 101.187,Z 70.000,A 180.000,B 0.000,C 180.000} C_DIS
LIN {X 66.031,Y 101.008,Z 70.000,A 180.000,B 0.000,C 180.000} C_DIS
LIN {X 65.999,Y 100.651,Z 70.000,A 180.000,B 0.000,C 180.000} C_DIS
LIN {X 65.980,Y 100.472,Z 70.000,A 180.000,B 0.000,C 180.000} C_DIS
LIN {X 65.969,Y 100.408,Z 70.000,A 180.000,B 0.000,C 180.000} C_DIS
LIN {X 65.949,Y 100.293,Z 70.000,A 180.000,B 0.000,C 180.000} C_DIS
LIN {X 65.917,Y 100.114,Z 70.000,A 180.000,B 0.000,C 180.000} C_DIS
LIN {X 65.885,Y 99.936,Z 70.000,A 180.000,B 0.000,C 180.000} C_DIS
LIN {X 65.845,Y 99.757,Z 70.000,A 180.000,B 0.000,C 180.000} C_DIS
LIN {X 65.796,Y 99.578,Z 70.000,A 180.000,B 0.000,C 180.000} C_DIS
LIN {X 65.748,Y 99.399,Z 70.000,A 180.000,B 0.000,C 180.000} C_DIS
LIN {X 65.698,Y 99.221,Z 70.000,A 180.000,B 0.000,C 180.000} C_DIS
LIN {X 65.635,Y 99.042,Z 70.000,A 180.000,B 0.000,C 180.000} C_DIS
LIN {X 65.503,Y 98.684,Z 70.000,A 180.000,B 0.000,C 180.000} C_DIS
LIN {X 65.433,Y 98.512,Z 70.000,A 180.000,B 0.000,C 180.000} C_DIS
LIN {X 65.430,Y 98.505,Z 70.000,A 180.000,B 0.000,C 180.000} C_DIS
LIN {X 65.346,Y 98.327,Z 70.000,A 180.000,B 0.000,C 180.000} C_DIS
LIN {X 65.254,Y 98.134,Z 70.000,A 180.000,B 0.000,C 180.000} C_DIS
LIN {X 65.174,Y 97.969,Z 70.000,A 180.000,B 0.000,C 180.000} C_DIS
LIN {X 65.075,Y 97.797,Z 70.000,A 180.000,B 0.000,C 180.000} C_DIS
LIN {X 64.897,Y 97.493,Z 70.000,A 180.000,B 0.000,C 180.000} C_DIS
LIN {X 64.861,Y 97.433,Z 70.000,A 180.000,B 0.000,C 180.000} C_DIS
LIN {X 64.739,Y 97.254,Z 70.000,A 180.000,B 0.000,C 180.000} C_DIS
LIN {X 64.539,Y 96.974,Z 70.000,A 180.000,B 0.000,C 180.000} C_DIS
LIN {X 64.484,Y 96.897,Z 70.000,A 180.000,B 0.000,C 180.000} C_DIS
LIN {X 64.360,Y 96.744,Z 70.000,A 180.000,B 0.000,C 180.000} C_DIS
LIN {X 64.182,Y 96.535,Z 70.000,A 180.000,B 0.000,C 180.000} C_DIS
LIN {X 64.030,Y 96.360,Z 70.000,A 180.000,B 0.000,C 180.000} C_DIS
LIN {X 64.003,Y 96.331,Z 70.000,A 180.000,B 0.000,C 180.000} C_DIS
LIN {X 63.853,Y 96.181,Z 70.000,A 180.000,B 0.000,C 180.000} C_DIS
LIN {X 63.645,Y 95.979,Z 70.000,A 180.000,B 0.000,C 180.000} C_DIS
LIN {X 63.477,Y 95.824,Z 70.000,A 180.000,B 0.000,C 180.000} C_DIS
LIN {X 63.467,Y 95.815,Z 70.000,A 180.000,B 0.000,C 180.000} C_DIS
LIN {X 63.288,Y 95.669,Z 70.000,A 180.000,B 0.000,C 180.000} C_DIS
LIN {X 63.109,Y 95.522,Z 70.000,A 180.000,B 0.000,C 180.000} C_DIS
LIN {X 63.038,Y 95.466,Z 70.000,A 180.000,B 0.000,C 180.000} C_DIS
LIN {X 62.930,Y 95.388,Z 70.000,A 180.000,B 0.000,C 180.000} C_DIS
LIN {X 62.573,Y 95.145,Z 70.000,A 180.000,B 0.000,C 180.000} C_DIS
LIN {X 62.518,Y 95.109,Z 70.000,A 180.000,B 0.000,C 180.000} C_DIS
LIN {X 62.394,Y 95.033,Z 70.000,A 180.000,B 0.000,C 180.000} C_DIS
LIN {X 62.210,Y 94.930,Z 70.000,A 180.000,B 0.000,C 180.000} C_DIS
LIN {X 62.036,Y 94.833,Z 70.000,A 180.000,B 0.000,C 180.000} C_DIS
LIN {X 61.885,Y 94.751,Z 70.000,A 180.000,B 0.000,C 180.000} C_DIS
LIN {X 61.858,Y 94.738,Z 70.000,A 180.000,B 0.000,C 180.000} C_DIS
LIN {X 61.679,Y 94.656,Z 70.000,A 180.000,B 0.000,C 180.000} C_DIS
LIN {X 61.491,Y 94.573,Z 70.000,A 180.000,B 0.000,C 180.000} C_DIS
LIN {X 61.321,Y 94.497,Z 70.000,A 180.000,B 0.000,C 180.000} C_DIS
LIN {X 61.143,Y 94.430,Z 70.000,A 180.000,B 0.000,C 180.000} C_DIS
LIN {X 60.785,Y 94.307,Z 70.000,A 180.000,B 0.000,C 180.000} C_DIS
LIN {X 60.606,Y 94.250,Z 70.000,A 180.000,B 0.000,C 180.000} C_DIS
LIN {X 60.470,Y 94.215,Z 70.000,A 180.000,B 0.000,C 180.000} C_DIS
LIN {X 60.249,Y 94.160,Z 70.000,A 180.000,B 0.000,C 180.000} C_DIS
LIN {X 60.070,Y 94.116,Z 70.000,A 180.000,B 0.000,C 180.000} C_DIS
LIN {X 59.891,Y 94.081,Z 70.000,A 180.000,B 0.000,C 180.000} C_DIS
LIN {X 59.534,Y 94.025,Z 70.000,A 180.000,B 0.000,C 180.000} C_DIS
LIN {X 59.355,Y 93.999,Z 70.000,A 180.000,B 0.000,C 180.000} C_DIS
LIN {X 59.176,Y 93.983,Z 70.000,A 180.000,B 0.000,C 180.000} C_DIS
LIN {X 58.819,Y 93.959,Z 70.000,A 180.000,B 0.000,C 180.000} C_DIS
LIN {X 58.640,Y 93.951,Z 70.000,A 180.000,B 0.000,C 180.000} C_DIS
LIN {X 58.461,Y 93.954,Z 70.000,A 180.000,B 0.000,C 180.000} C_DIS
LIN {X 58.103,Y 93.962,Z 70.000,A 180.000,B 0.000,C 180.000} C_DIS
LIN {X 57.925,Y 93.973,Z 70.000,A 180.000,B 0.000,C 180.000} C_DIS
LIN {X 57.746,Y 93.992,Z 70.000,A 180.000,B 0.000,C 180.000} C_DIS
LIN {X 57.567,Y 94.012,Z 70.000,A 180.000,B 0.000,C 180.000} C_DIS
LIN {X 57.388,Y 94.033,Z 70.000,A 180.000,B 0.000,C 180.000} C_DIS
LIN {X 57.363,Y 94.036,Z 70.000,A 180.000,B 0.000,C 180.000} C_DIS
LIN {X 57.210,Y 94.063,Z 70.000,A 180.000,B 0.000,C 180.000} C_DIS
LIN {X 56.852,Y 94.135,Z 70.000,A 180.000,B 0.000,C 180.000} C_DIS
LIN {X 56.673,Y 94.174,Z 70.000,A 180.000,B 0.000,C 180.000} C_DIS
LIN {X 56.528,Y 94.215,Z 70.000,A 180.000,B 0.000,C 180.000} C_DIS
LIN {X 56.316,Y 94.278,Z 70.000,A 180.000,B 0.000,C 180.000} C_DIS
LIN {X 56.137,Y 94.331,Z 70.000,A 180.000,B 0.000,C 180.000} C_DIS
LIN {X 55.958,Y 94.392,Z 70.000,A 180.000,B 0.000,C 180.000} C_DIS
LIN {X 55.953,Y 94.394,Z 70.000,A 180.000,B 0.000,C 180.000} C_DIS
LIN {X 55.779,Y 94.462,Z 70.000,A 180.000,B 0.000,C 180.000} C_DIS
LIN {X 55.601,Y 94.533,Z 70.000,A 180.000,B 0.000,C 180.000} C_DIS
LIN {X 55.501,Y 94.573,Z 70.000,A 180.000,B 0.000,C 180.000} C_DIS
LIN {X 55.422,Y 94.606,Z 70.000,A 180.000,B 0.000,C 180.000} C_DIS
LIN {X 55.243,Y 94.693,Z 70.000,A 180.000,B 0.000,C 180.000} C_DIS
LIN {X 55.064,Y 94.782,Z 70.000,A 180.000,B 0.000,C 180.000} C_DIS
LIN {X 54.886,Y 94.872,Z 70.000,A 180.000,B 0.000,C 180.000} C_DIS
LIN {X 54.781,Y 94.930,Z 70.000,A 180.000,B 0.000,C 180.000} C_DIS
LIN {X 54.707,Y 94.975,Z 70.000,A 180.000,B 0.000,C 180.000} C_DIS
LIN {X 54.349,Y 95.195,Z 70.000,A 180.000,B 0.000,C 180.000} C_DIS
LIN {X 54.210,Y 95.288,Z 70.000,A 180.000,B 0.000,C 180.000} C_DIS
LIN {X 54.177,Y 95.312,Z 70.000,A 180.000,B 0.000,C 180.000} C_DIS
LIN {X 54.171,Y 95.316,Z 70.000,A 180.000,B 0.000,C 180.000} C_DIS
LIN {X 53.970,Y 95.466,Z 70.000,A 180.000,B 0.000,C 180.000} C_DIS
LIN {X 53.813,Y 95.583,Z 70.000,A 180.000,B 0.000,C 180.000} C_DIS
LIN {X 53.733,Y 95.645,Z 70.000,A 180.000,B 0.000,C 180.000} C_DIS
LIN {X 53.634,Y 95.729,Z 70.000,A 180.000,B 0.000,C 180.000} C_DIS
LIN {X 53.329,Y 96.003,Z 70.000,A 180.000,B 0.000,C 180.000} C_DIS
LIN {X 53.277,Y 96.050,Z 70.000,A 180.000,B 0.000,C 180.000} C_DIS
LIN {X 53.144,Y 96.181,Z 70.000,A 180.000,B 0.000,C 180.000} C_DIS
LIN {X 52.919,Y 96.421,Z 70.000,A 180.000,B 0.000,C 180.000} C_DIS
LIN {X 52.810,Y 96.539,Z 70.000,A 180.000,B 0.000,C 180.000} C_DIS
LIN {X 52.740,Y 96.619,Z 70.000,A 180.000,B 0.000,C 180.000} C_DIS
LIN {X 52.662,Y 96.718,Z 70.000,A 180.000,B 0.000,C 180.000} C_DIS
LIN {X 52.522,Y 96.897,Z 70.000,A 180.000,B 0.000,C 180.000} C_DIS
LIN {X 52.383,Y 97.075,Z 70.000,A 180.000,B 0.000,C 180.000} C_DIS
LIN {X 52.261,Y 97.254,Z 70.000,A 180.000,B 0.000,C 180.000} C_DIS
LIN {X 52.145,Y 97.433,Z 70.000,A 180.000,B 0.000,C 180.000} C_DIS
LIN {X 52.029,Y 97.612,Z 70.000,A 180.000,B 0.000,C 180.000} C_DIS
LIN {X 52.025,Y 97.618,Z 70.000,A 180.000,B 0.000,C 180.000} C_DIS
LIN {X 51.927,Y 97.790,Z 70.000,A 180.000,B 0.000,C 180.000} C_DIS
LIN {X 51.737,Y 98.148,Z 70.000,A 180.000,B 0.000,C 180.000} C_DIS
LIN {X 51.668,Y 98.287,Z 70.000,A 180.000,B 0.000,C 180.000} C_DIS
LIN {X 51.650,Y 98.327,Z 70.000,A 180.000,B 0.000,C 180.000} C_DIS
LIN {X 51.574,Y 98.505,Z 70.000,A 180.000,B 0.000,C 180.000} C_DIS
LIN {X 51.489,Y 98.708,Z 70.000,A 180.000,B 0.000,C 180.000} C_DIS
LIN {X 51.426,Y 98.863,Z 70.000,A 180.000,B 0.000,C 180.000} C_DIS
LIN {X 51.365,Y 99.042,Z 70.000,A 180.000,B 0.000,C 180.000} C_DIS
LIN {X 51.250,Y 99.399,Z 70.000,A 180.000,B 0.000,C 180.000} C_DIS
LIN {X 51.199,Y 99.578,Z 70.000,A 180.000,B 0.000,C 180.000} C_DIS
LIN {X 51.159,Y 99.757,Z 70.000,A 180.000,B 0.000,C 180.000} C_DIS
LIN {X 51.118,Y 99.936,Z 70.000,A 180.000,B 0.000,C 180.000} C_DIS
LIN {X 51.079,Y 100.114,Z 70.000,A 180.000,B 0.000,C 180.000} C_DIS
LIN {X 51.049,Y 100.293,Z 70.000,A 180.000,B 0.000,C 180.000} C_DIS
LIN {X 51.001,Y 100.651,Z 70.000,A 180.000,B 0.000,C 180.000} C_DIS
LIN {X 50.980,Y 100.829,Z 70.000,A 180.000,B 0.000,C 180.000} C_DIS
LIN {X 50.969,Y 101.008,Z 70.000,A 180.000,B 0.000,C 180.000} C_DIS
LIN {X 50.953,Y 101.385,Z 70.000,A 180.000,B 0.000,C 180.000} C_DIS
LIN {X 50.950,Y 101.545,Z 70.000,A 180.000,B 0.000,C 180.000} C_DIS
LIN {X 50.953,Y 101.615,Z 70.000,A 180.000,B 0.000,C 180.000} C_DIS
LIN {X 50.965,Y 101.902,Z 70.000,A 180.000,B 0.000,C 180.000} C_DIS
LIN {X 50.973,Y 102.081,Z 70.000,A 180.000,B 0.000,C 180.000} C_DIS
LIN {X 50.989,Y 102.260,Z 70.000,A 180.000,B 0.000,C 180.000} C_DIS
LIN {X 51.013,Y 102.438,Z 70.000,A 180.000,B 0.000,C 180.000} C_DIS
LIN {X 51.037,Y 102.617,Z 70.000,A 180.000,B 0.000,C 180.000} C_DIS
LIN {X 51.062,Y 102.796,Z 70.000,A 180.000,B 0.000,C 180.000} C_DIS
LIN {X 51.098,Y 102.975,Z 70.000,A 180.000,B 0.000,C 180.000} C_DIS
LIN {X 51.179,Y 103.332,Z 70.000,A 180.000,B 0.000,C 180.000} C_DIS
LIN {X 51.188,Y 103.372,Z 70.000,A 180.000,B 0.000,C 180.000} C_DIS
; Lead Out Move Starts
LIN {X 51.131,Y 103.750,Z 70.000,A 180.000,B 0.000,C 180.000} C_DIS
LIN {X 50.823,Y 103.977,Z 70.000,A 180.000,B 0.000,C 180.000} C_DIS
; Link Move Starts
LIN {X 50.707,Y 104.022,Z 70.000,A 180.000,B 0.000,C 180.000} C_DIS
LIN {X 44.913,Y 107.136,Z 70.000,A 180.000,B 0.000,C 180.000} C_DIS
LIN {X 43.634,Y 107.414,Z 70.000,A 180.000,B 0.000,C 180.000} C_DIS
LIN {X 42.402,Y 106.972,Z 70.000,A 180.000,B 0.000,C 180.000} C_DIS
LIN {X 41.591,Y 105.945,Z 70.000,A 180.000,B 0.000,C 180.000} C_DIS
LIN {X 41.448,Y 104.644,Z 70.000,A 180.000,B 0.000,C 180.000} C_DIS
LIN {X 42.016,Y 103.464,Z 70.000,A 180.000,B 0.000,C 180.000} C_DIS
LIN {X 43.122,Y 102.765,Z 70.000,A 180.000,B 0.000,C 180.000} C_DIS
LIN {X 44.431,Y 102.758,Z 70.000,A 180.000,B 0.000,C 180.000} C_DIS
$VEL.CP=0.01
LIN {X 44.448,Y 102.763,Z 70.000,A 180.000,B 0.000,C 180.000} C_DIS
LIN {X 45.581,Y 103.486,Z 69.952,A 180.000,B 0.000,C 180.000} C_DIS
LIN {X 46.140,Y 104.709,Z 69.905,A 180.000,B 0.000,C 180.000} C_DIS
LIN {X 45.945,Y 106.040,Z 69.857,A 180.000,B 0.000,C 180.000} C_DIS
LIN {X 45.059,Y 107.051,Z 69.809,A 180.000,B 0.000,C 180.000} C_DIS
LIN {X 43.766,Y 107.419,Z 69.762,A 180.000,B 0.000,C 180.000} C_DIS
LIN {X 42.480,Y 107.026,Z 69.714,A 180.000,B 0.000,C 180.000} C_DIS
LIN {X 41.614,Y 105.997,Z 69.667,A 180.000,B 0.000,C 180.000} C_DIS
LIN {X 41.445,Y 104.663,Z 69.619,A 180.000,B 0.000,C 180.000} C_DIS
LIN {X 42.027,Y 103.451,Z 69.571,A 180.000,B 0.000,C 180.000} C_DIS
LIN {X 43.175,Y 102.750,Z 69.524,A 180.000,B 0.000,C 180.000} C_DIS
LIN {X 44.519,Y 102.784,Z 69.476,A 180.000,B 0.000,C 180.000} C_DIS
LIN {X 45.629,Y 103.543,Z 69.429,A 180.000,B 0.000,C 180.000} C_DIS
LIN {X 46.150,Y 104.783,Z 69.381,A 180.000,B 0.000,C 180.000} C_DIS
LIN {X 45.913,Y 106.107,Z 69.333,A 180.000,B 0.000,C 180.000} C_DIS
LIN {X 44.996,Y 107.090,Z 69.286,A 180.000,B 0.000,C 180.000} C_DIS
LIN {X 43.691,Y 107.417,Z 69.238,A 180.000,B 0.000,C 180.000} C_DIS
LIN {X 42.418,Y 106.984,Z 69.191,A 180.000,B 0.000,C 180.000} C_DIS
LIN {X 41.585,Y 105.929,Z 69.143,A 180.000,B 0.000,C 180.000} C_DIS
LIN {X 41.458,Y 104.590,Z 69.095,A 180.000,B 0.000,C 180.000} C_DIS
LIN {X 42.078,Y 103.397,Z 69.048,A 180.000,B 0.000,C 180.000} C_DIS
LIN {X 43.247,Y 102.732,Z 69.000,A 180.000,B 0.000,C 180.000} C_DIS
LIN {X 43.264,Y 102.728,Z 69.000,A 180.000,B 0.000,C 180.000} C_DIS
; Lead In Move Starts
LIN {X 43.513,Y 102.672,Z 69.000,A 180.000,B 0.000,C 180.000} C_DIS
LIN {X 44.744,Y 102.720,Z 69.000,A 180.000,B 0.000,C 180.000} C_DIS
LIN {X 45.786,Y 103.376,Z 69.000,A 180.000,B 0.000,C 180.000} C_DIS
LIN {X 46.360,Y 104.467,Z 69.000,A 180.000,B 0.000,C 180.000} C_DIS
; Cutting Move Starts
$VEL.CP=0.02
LIN {X 46.386,Y 104.584,Z 69.000,A 180.000,B 0.000,C 180.000} C_DIS
LIN {X 46.436,Y 104.762,Z 69.000,A 180.000,B 0.000,C 180.000} C_DIS
LIN {X 46.540,Y 105.120,Z 69.000,A 180.000,B 0.000,C 180.000} C_DIS
LIN {X 46.592,Y 105.299,Z 69.000,A 180.000,B 0.000,C 180.000} C_DIS
LIN {X 46.652,Y 105.477,Z 69.000,A 180.000,B 0.000,C 180.000} C_DIS
LIN {X 46.845,Y 106.014,Z 69.000,A 180.000,B 0.000,C 180.000} C_DIS
LIN {X 46.916,Y 106.193,Z 69.000,A 180.000,B 0.000,C 180.000} C_DIS
LIN {X 47.148,Y 106.729,Z 69.000,A 180.000,B 0.000,C 180.000} C_DIS
LIN {X 47.198,Y 106.841,Z 69.000,A 180.000,B 0.000,C 180.000} C_DIS
LIN {X 47.232,Y 106.908,Z 69.000,A 180.000,B 0.000,C 180.000} C_DIS
LIN {X 47.505,Y 107.444,Z 69.000,A 180.000,B 0.000,C 180.000} C_DIS
LIN {X 47.556,Y 107.540,Z 69.000,A 180.000,B 0.000,C 180.000} C_DIS
LIN {X 47.604,Y 107.623,Z 69.000,A 180.000,B 0.000,C 180.000} C_DIS
LIN {X 47.816,Y 107.980,Z 69.000,A 180.000,B 0.000,C 180.000} C_DIS
LIN {X 47.914,Y 108.145,Z 69.000,A 180.000,B 0.000,C 180.000} C_DIS
LIN {X 47.922,Y 108.159,Z 69.000,A 180.000,B 0.000,C 180.000} C_DIS
LIN {X 48.040,Y 108.338,Z 69.000,A 180.000,B 0.000,C 180.000} C_DIS
LIN {X 48.283,Y 108.695,Z 69.000,A 180.000,B 0.000,C 180.000} C_DIS
LIN {X 48.407,Y 108.874,Z 69.000,A 180.000,B 0.000,C 180.000} C_DIS
LIN {X 48.450,Y 108.930,Z 69.000,A 180.000,B 0.000,C 180.000} C_DIS
LIN {X 48.823,Y 109.410,Z 69.000,A 180.000,B 0.000,C 180.000} C_DIS
LIN {X 48.974,Y 109.589,Z 69.000,A 180.000,B 0.000,C 180.000} C_DIS
LIN {X 49.289,Y 109.947,Z 69.000,A 180.000,B 0.000,C 180.000} C_DIS
LIN {X 49.344,Y 110.009,Z 69.000,A 180.000,B 0.000,C 180.000} C_DIS
LIN {X 49.455,Y 110.126,Z 69.000,A 180.000,B 0.000,C 180.000} C_DIS
LIN {X 49.880,Y 110.551,Z 69.000,A 180.000,B 0.000,C 180.000} C_DIS
LIN {X 49.998,Y 110.662,Z 69.000,A 180.000,B 0.000,C 180.000} C_DIS
LIN {X 50.416,Y 111.031,Z 69.000,A 180.000,B 0.000,C 180.000} C_DIS
LIN {X 50.595,Y 111.182,Z 69.000,A 180.000,B 0.000,C 180.000} C_DIS
LIN {X 51.077,Y 111.556,Z 69.000,A 180.000,B 0.000,C 180.000} C_DIS
LIN {X 51.131,Y 111.597,Z 69.000,A 180.000,B 0.000,C 180.000} C_DIS
LIN {X 51.310,Y 111.721,Z 69.000,A 180.000,B 0.000,C 180.000} C_DIS
LIN {X 51.668,Y 111.964,Z 69.000,A 180.000,B 0.000,C 180.000} C_DIS
LIN {X 51.847,Y 112.082,Z 69.000,A 180.000,B 0.000,C 180.000} C_DIS
LIN {X 51.864,Y 112.092,Z 69.000,A 180.000,B 0.000,C 180.000} C_DIS
LIN {X 52.204,Y 112.293,Z 69.000,A 180.000,B 0.000,C 180.000} C_DIS
LIN {X 52.383,Y 112.399,Z 69.000,A 180.000,B 0.000,C 180.000} C_DIS
LIN {X 52.470,Y 112.450,Z 69.000,A 180.000,B 0.000,C 180.000} C_DIS
LIN {X 52.562,Y 112.498,Z 69.000,A 180.000,B 0.000,C 180.000} C_DIS
LIN {X 53.098,Y 112.771,Z 69.000,A 180.000,B 0.000,C 180.000} C_DIS
LIN {X 53.171,Y 112.807,Z 69.000,A 180.000,B 0.000,C 180.000} C_DIS
LIN {X 53.277,Y 112.854,Z 69.000,A 180.000,B 0.000,C 180.000} C_DIS
LIN {X 53.813,Y 113.087,Z 69.000,A 180.000,B 0.000,C 180.000} C_DIS
LIN {X 53.992,Y 113.157,Z 69.000,A 180.000,B 0.000,C 180.000} C_DIS
LIN {X 54.528,Y 113.350,Z 69.000,A 180.000,B 0.000,C 180.000} C_DIS
LIN {X 54.707,Y 113.410,Z 69.000,A 180.000,B 0.000,C 180.000} C_DIS
LIN {X 55.243,Y 113.566,Z 69.000,A 180.000,B 0.000,C 180.000} C_DIS
LIN {X 55.422,Y 113.615,Z 69.000,A 180.000,B 0.000,C 180.000} C_DIS
LIN {X 55.601,Y 113.655,Z 69.000,A 180.000,B 0.000,C 180.000} C_DIS
LIN {X 55.958,Y 113.735,Z 69.000,A 180.000,B 0.000,C 180.000} C_DIS
LIN {X 56.137,Y 113.775,Z 69.000,A 180.000,B 0.000,C 180.000} C_DIS
LIN {X 56.316,Y 113.805,Z 69.000,A 180.000,B 0.000,C 180.000} C_DIS
LIN {X 56.852,Y 113.890,Z 69.000,A 180.000,B 0.000,C 180.000} C_DIS
LIN {X 57.031,Y 113.912,Z 69.000,A 180.000,B 0.000,C 180.000} C_DIS
LIN {X 57.567,Y 113.963,Z 69.000,A 180.000,B 0.000,C 180.000} C_DIS
LIN {X 57.746,Y 113.977,Z 69.000,A 180.000,B 0.000,C 180.000} C_DIS
LIN {X 57.925,Y 113.983,Z 69.000,A 180.000,B 0.000,C 180.000} C_DIS
LIN {X 58.282,Y 113.994,Z 69.000,A 180.000,B 0.000,C 180.000} C_DIS
LIN {X 58.461,Y 114.000,Z 69.000,A 180.000,B 0.000,C 180.000} C_DIS
LIN {X 58.640,Y 113.997,Z 69.000,A 180.000,B 0.000,C 180.000} C_DIS
LIN {X 59.176,Y 113.980,Z 69.000,A 180.000,B 0.000,C 180.000} C_DIS
LIN {X 59.355,Y 113.970,Z 69.000,A 180.000,B 0.000,C 180.000} C_DIS
LIN {X 59.534,Y 113.953,Z 69.000,A 180.000,B 0.000,C 180.000} C_DIS
LIN {X 59.891,Y 113.919,Z 69.000,A 180.000,B 0.000,C 180.000} C_DIS
LIN {X 60.070,Y 113.901,Z 69.000,A 180.000,B 0.000,C 180.000} C_DIS
LIN {X 60.212,Y 113.880,Z 69.000,A 180.000,B 0.000,C 180.000} C_DIS
LIN {X 60.606,Y 113.817,Z 69.000,A 180.000,B 0.000,C 180.000} C_DIS
LIN {X 60.785,Y 113.789,Z 69.000,A 180.000,B 0.000,C 180.000} C_DIS
LIN {X 60.964,Y 113.753,Z 69.000,A 180.000,B 0.000,C 180.000} C_DIS
LIN {X 61.500,Y 113.633,Z 69.000,A 180.000,B 0.000,C 180.000} C_DIS
LIN {X 61.679,Y 113.588,Z 69.000,A 180.000,B 0.000,C 180.000} C_DIS
LIN {X 62.215,Y 113.432,Z 69.000,A 180.000,B 0.000,C 180.000} C_DIS
LIN {X 62.394,Y 113.378,Z 69.000,A 180.000,B 0.000,C 180.000} C_DIS
LIN {X 62.491,Y 113.343,Z 69.000,A 180.000,B 0.000,C 180.000} C_DIS
LIN {X 62.987,Y 113.165,Z 69.000,A 180.000,B 0.000,C 180.000} C_DIS
LIN {X 63.109,Y 113.119,Z 69.000,A 180.000,B 0.000,C 180.000} C_DIS
LIN {X 63.288,Y 113.043,Z 69.000,A 180.000,B 0.000,C 180.000} C_DIS
LIN {X 63.645,Y 112.888,Z 69.000,A 180.000,B 0.000,C 180.000} C_DIS
LIN {X 63.824,Y 112.809,Z 69.000,A 180.000,B 0.000,C 180.000} C_DIS
LIN {X 63.829,Y 112.807,Z 69.000,A 180.000,B 0.000,C 180.000} C_DIS
LIN {X 64.003,Y 112.720,Z 69.000,A 180.000,B 0.000,C 180.000} C_DIS
LIN {X 64.360,Y 112.538,Z 69.000,A 180.000,B 0.000,C 180.000} C_DIS
LIN {X 64.530,Y 112.450,Z 69.000,A 180.000,B 0.000,C 180.000} C_DIS
LIN {X 64.539,Y 112.444,Z 69.000,A 180.000,B 0.000,C 180.000} C_DIS
LIN {X 64.718,Y 112.339,Z 69.000,A 180.000,B 0.000,C 180.000} C_DIS
LIN {X 65.075,Y 112.128,Z 69.000,A 180.000,B 0.000,C 180.000} C_DIS
LIN {X 65.136,Y 112.092,Z 69.000,A 180.000,B 0.000,C 180.000} C_DIS
LIN {X 65.254,Y 112.017,Z 69.000,A 180.000,B 0.000,C 180.000} C_DIS
LIN {X 65.433,Y 111.896,Z 69.000,A 180.000,B 0.000,C 180.000} C_DIS
LIN {X 65.670,Y 111.734,Z 69.000,A 180.000,B 0.000,C 180.000} C_DIS
LIN {X 65.791,Y 111.653,Z 69.000,A 180.000,B 0.000,C 180.000} C_DIS
LIN {X 65.923,Y 111.556,Z 69.000,A 180.000,B 0.000,C 180.000} C_DIS
LIN {X 66.384,Y 111.198,Z 69.000,A 180.000,B 0.000,C 180.000} C_DIS
LIN {X 66.506,Y 111.099,Z 69.000,A 180.000,B 0.000,C 180.000} C_DIS
LIN {X 66.597,Y 111.019,Z 69.000,A 180.000,B 0.000,C 180.000} C_DIS
LIN {X 67.002,Y 110.662,Z 69.000,A 180.000,B 0.000,C 180.000} C_DIS
LIN {X 67.042,Y 110.626,Z 69.000,A 180.000,B 0.000,C 180.000} C_DIS
LIN {X 67.188,Y 110.483,Z 69.000,A 180.000,B 0.000,C 180.000} C_DIS
LIN {X 67.545,Y 110.126,Z 69.000,A 180.000,B 0.000,C 180.000} C_DIS
LIN {X 67.578,Y 110.092,Z 69.000,A 180.000,B 0.000,C 180.000} C_DIS
LIN {X 67.711,Y 109.947,Z 69.000,A 180.000,B 0.000,C 180.000} C_DIS
LIN {X 68.026,Y 109.589,Z 69.000,A 180.000,B 0.000,C 180.000} C_DIS
LIN {X 68.115,Y 109.488,Z 69.000,A 180.000,B 0.000,C 180.000} C_DIS
LIN {X 68.177,Y 109.410,Z 69.000,A 180.000,B 0.000,C 180.000} C_DIS
LIN {X 68.472,Y 109.031,Z 69.000,A 180.000,B 0.000,C 180.000} C_DIS
LIN {X 68.593,Y 108.874,Z 69.000,A 180.000,B 0.000,C 180.000} C_DIS
LIN {X 68.651,Y 108.793,Z 69.000,A 180.000,B 0.000,C 180.000} C_DIS
LIN {X 68.717,Y 108.695,Z 69.000,A 180.000,B 0.000,C 180.000} C_DIS
LIN {X 69.008,Y 108.267,Z 69.000,A 180.000,B 0.000,C 180.000} C_DIS
LIN {X 69.078,Y 108.159,Z 69.000,A 180.000,B 0.000,C 180.000} C_DIS
LIN {X 69.184,Y 107.980,Z 69.000,A 180.000,B 0.000,C 180.000} C_DIS
LIN {X 69.396,Y 107.623,Z 69.000,A 180.000,B 0.000,C 180.000} C_DIS
LIN {X 69.495,Y 107.444,Z 69.000,A 180.000,B 0.000,C 180.000} C_DIS
LIN {X 69.768,Y 106.908,Z 69.000,A 180.000,B 0.000,C 180.000} C_DIS
LIN {X 69.852,Y 106.729,Z 69.000,A 180.000,B 0.000,C 180.000} C_DIS
LIN {X 70.084,Y 106.193,Z 69.000,A 180.000,B 0.000,C 180.000} C_DIS
LIN {X 70.155,Y 106.014,Z 69.000,A 180.000,B 0.000,C 180.000} C_DIS
LIN {X 70.348,Y 105.477,Z 69.000,A 180.000,B 0.000,C 180.000} C_DIS
LIN {X 70.408,Y 105.299,Z 69.000,A 180.000,B 0.000,C 180.000} C_DIS
LIN {X 70.439,Y 105.194,Z 69.000,A 180.000,B 0.000,C 180.000} C_DIS
LIN {X 70.564,Y 104.762,Z 69.000,A 180.000,B 0.000,C 180.000} C_DIS
LIN {X 70.614,Y 104.584,Z 69.000,A 180.000,B 0.000,C 180.000} C_DIS
LIN {X 70.617,Y 104.568,Z 69.000,A 180.000,B 0.000,C 180.000} C_DIS
LIN {X 70.654,Y 104.405,Z 69.000,A 180.000,B 0.000,C 180.000} C_DIS
LIN {X 70.734,Y 104.047,Z 69.000,A 180.000,B 0.000,C 180.000} C_DIS
LIN {X 70.773,Y 103.869,Z 69.000,A 180.000,B 0.000,C 180.000} C_DIS
LIN {X 70.796,Y 103.739,Z 69.000,A 180.000,B 0.000,C 180.000} C_DIS
LIN {X 70.889,Y 103.153,Z 69.000,A 180.000,B 0.000,C 180.000} C_DIS
LIN {X 70.911,Y 102.975,Z 69.000,A 180.000,B 0.000,C 180.000} C_DIS
LIN {X 70.962,Y 102.438,Z 69.000,A 180.000,B 0.000,C 180.000} C_DIS
LIN {X 70.975,Y 102.292,Z 69.000,A 180.000,B 0.000,C 180.000} C_DIS
LIN {X 70.977,Y 102.260,Z 69.000,A 180.000,B 0.000,C 180.000} C_DIS
LIN {X 70.983,Y 102.081,Z 69.000,A 180.000,B 0.000,C 180.000} C_DIS
LIN {X 70.994,Y 101.723,Z 69.000,A 180.000,B 0.000,C 180.000} C_DIS
LIN {X 71.000,Y 101.545,Z 69.000,A 180.000,B 0.000,C 180.000} C_DIS
LIN {X 70.997,Y 101.366,Z 69.000,A 180.000,B 0.000,C 180.000} C_DIS
LIN {X 70.980,Y 100.829,Z 69.000,A 180.000,B 0.000,C 180.000} C_DIS
LIN {X 70.975,Y 100.708,Z 69.000,A 180.000,B 0.000,C 180.000} C_DIS
LIN {X 70.970,Y 100.651,Z 69.000,A 180.000,B 0.000,C 180.000} C_DIS
LIN {X 70.954,Y 100.472,Z 69.000,A 180.000,B 0.000,C 180.000} C_DIS
LIN {X 70.920,Y 100.114,Z 69.000,A 180.000,B 0.000,C 180.000} C_DIS
LIN {X 70.902,Y 99.936,Z 69.000,A 180.000,B 0.000,C 180.000} C_DIS
LIN {X 70.875,Y 99.757,Z 69.000,A 180.000,B 0.000,C 180.000} C_DIS
LIN {X 70.796,Y 99.261,Z 69.000,A 180.000,B 0.000,C 180.000} C_DIS
LIN {X 70.790,Y 99.221,Z 69.000,A 180.000,B 0.000,C 180.000} C_DIS
LIN {X 70.754,Y 99.042,Z 69.000,A 180.000,B 0.000,C 180.000} C_DIS
LIN {X 70.670,Y 98.665,Z 69.000,A 180.000,B 0.000,C 180.000} C_DIS
LIN {X 70.634,Y 98.505,Z 69.000,A 180.000,B 0.000,C 180.000} C_DIS
LIN {X 70.617,Y 98.432,Z 69.000,A 180.000,B 0.000,C 180.000} C_DIS
LIN {X 70.590,Y 98.327,Z 69.000,A 180.000,B 0.000,C 180.000} C_DIS
LIN {X 70.538,Y 98.148,Z 69.000,A 180.000,B 0.000,C 180.000} C_DIS
LIN {X 70.434,Y 97.790,Z 69.000,A 180.000,B 0.000,C 180.000} C_DIS
LIN {X 70.380,Y 97.612,Z 69.000,A 180.000,B 0.000,C 180.000} C_DIS
LIN {X 70.316,Y 97.433,Z 69.000,A 180.000,B 0.000,C 180.000} C_DIS
LIN {X 70.187,Y 97.075,Z 69.000,A 180.000,B 0.000,C 180.000} C_DIS
LIN {X 70.121,Y 96.897,Z 69.000,A 180.000,B 0.000,C 180.000} C_DIS
LIN {X 70.081,Y 96.800,Z 69.000,A 180.000,B 0.000,C 180.000} C_DIS
LIN {X 69.891,Y 96.360,Z 69.000,A 180.000,B 0.000,C 180.000} C_DIS
LIN {X 69.812,Y 96.181,Z 69.000,A 180.000,B 0.000,C 180.000} C_DIS
LIN {X 69.724,Y 96.005,Z 69.000,A 180.000,B 0.000,C 180.000} C_DIS
LIN {X 69.540,Y 95.645,Z 69.000,A 180.000,B 0.000,C 180.000} C_DIS
LIN {X 69.447,Y 95.466,Z 69.000,A 180.000,B 0.000,C 180.000} C_DIS
LIN {X 69.366,Y 95.327,Z 69.000,A 180.000,B 0.000,C 180.000} C_DIS
LIN {X 69.131,Y 94.930,Z 69.000,A 180.000,B 0.000,C 180.000} C_DIS
LIN {X 69.021,Y 94.751,Z 69.000,A 180.000,B 0.000,C 180.000} C_DIS
LIN {X 69.008,Y 94.733,Z 69.000,A 180.000,B 0.000,C 180.000} C_DIS
LIN {X 68.657,Y 94.215,Z 69.000,A 180.000,B 0.000,C 180.000} C_DIS
LIN {X 68.651,Y 94.207,Z 69.000,A 180.000,B 0.000,C 180.000} C_DIS
LIN {X 68.524,Y 94.036,Z 69.000,A 180.000,B 0.000,C 180.000} C_DIS
LIN {X 68.247,Y 93.679,Z 69.000,A 180.000,B 0.000,C 180.000} C_DIS
LIN {X 68.115,Y 93.512,Z 69.000,A 180.000,B 0.000,C 180.000} C_DIS
LIN {X 68.104,Y 93.500,Z 69.000,A 180.000,B 0.000,C 180.000} C_DIS
LIN {X 67.947,Y 93.321,Z 69.000,A 180.000,B 0.000,C 180.000} C_DIS
LIN {X 67.757,Y 93.106,Z 69.000,A 180.000,B 0.000,C 180.000} C_DIS
LIN {X 67.631,Y 92.964,Z 69.000,A 180.000,B 0.000,C 180.000} C_DIS
LIN {X 67.578,Y 92.908,Z 69.000,A 180.000,B 0.000,C 180.000} C_DIS
LIN {X 67.456,Y 92.785,Z 69.000,A 180.000,B 0.000,C 180.000} C_DIS
LIN {X 67.221,Y 92.550,Z 69.000,A 180.000,B 0.000,C 180.000} C_DIS
LIN {X 67.098,Y 92.427,Z 69.000,A 180.000,B 0.000,C 180.000} C_DIS
LIN {X 67.042,Y 92.374,Z 69.000,A 180.000,B 0.000,C 180.000} C_DIS
LIN {X 66.901,Y 92.249,Z 69.000,A 180.000,B 0.000,C 180.000} C_DIS
LIN {X 66.684,Y 92.058,Z 69.000,A 180.000,B 0.000,C 180.000} C_DIS
LIN {X 66.506,Y 91.901,Z 69.000,A 180.000,B 0.000,C 180.000} C_DIS
LIN {X 66.494,Y 91.891,Z 69.000,A 180.000,B 0.000,C 180.000} C_DIS
LIN {X 66.327,Y 91.758,Z 69.000,A 180.000,B 0.000,C 180.000} C_DIS
LIN {X 65.969,Y 91.480,Z 69.000,A 180.000,B 0.000,C 180.000} C_DIS
LIN {X 65.801,Y 91.355,Z 69.000,A 180.000,B 0.000,C 180.000} C_DIS
LIN {X 65.791,Y 91.347,Z 69.000,A 180.000,B 0.000,C 180.000} C_DIS
LIN {X 65.538,Y 91.176,Z 69.000,A 180.000,B 0.000,C 180.000} C_DIS
LIN {X 65.275,Y 90.997,Z 69.000,A 180.000,B 0.000,C 180.000} C_DIS
LIN {X 65.254,Y 90.983,Z 69.000,A 180.000,B 0.000,C 180.000} C_DIS
LIN {X 65.075,Y 90.872,Z 69.000,A 180.000,B 0.000,C 180.000} C_DIS
LIN {X 64.682,Y 90.640,Z 69.000,A 180.000,B 0.000,C 180.000} C_DIS
LIN {X 64.539,Y 90.556,Z 69.000,A 180.000,B 0.000,C 180.000} C_DIS
LIN {X 64.360,Y 90.462,Z 69.000,A 180.000,B 0.000,C 180.000} C_DIS
LIN {X 64.003,Y 90.280,Z 69.000,A 180.000,B 0.000,C 180.000} C_DIS
LIN {X 63.824,Y 90.191,Z 69.000,A 180.000,B 0.000,C 180.000} C_DIS
LIN {X 63.645,Y 90.112,Z 69.000,A 180.000,B 0.000,C 180.000} C_DIS
LIN {X 63.213,Y 89.925,Z 69.000,A 180.000,B 0.000,C 180.000} C_DIS
LIN {X 63.109,Y 89.881,Z 69.000,A 180.000,B 0.000,C 180.000} C_DIS
LIN {X 62.930,Y 89.815,Z 69.000,A 180.000,B 0.000,C 180.000} C_DIS
LIN {X 62.573,Y 89.686,Z 69.000,A 180.000,B 0.000,C 180.000} C_DIS
LIN {X 62.394,Y 89.622,Z 69.000,A 180.000,B 0.000,C 180.000} C_DIS
LIN {X 62.215,Y 89.568,Z 69.000,A 180.000,B 0.000,C 180.000} C_DIS
LIN {X 61.679,Y 89.412,Z 69.000,A 180.000,B 0.000,C 180.000} C_DIS
LIN {X 61.591,Y 89.388,Z 69.000,A 180.000,B 0.000,C 180.000} C_DIS
LIN {X 61.500,Y 89.367,Z 69.000,A 180.000,B 0.000,C 180.000} C_DIS
LIN {X 60.964,Y 89.247,Z 69.000,A 180.000,B 0.000,C 180.000} C_DIS
LIN {X 60.785,Y 89.211,Z 69.000,A 180.000,B 0.000,C 180.000} C_DIS
LIN {X 60.774,Y 89.209,Z 69.000,A 180.000,B 0.000,C 180.000} C_DIS
LIN {X 60.606,Y 89.183,Z 69.000,A 180.000,B 0.000,C 180.000} C_DIS
LIN {X 60.249,Y 89.126,Z 69.000,A 180.000,B 0.000,C 180.000} C_DIS
LIN {X 60.070,Y 89.099,Z 69.000,A 180.000,B 0.000,C 180.000} C_DIS
LIN {X 59.891,Y 89.081,Z 69.000,A 180.000,B 0.000,C 180.000} C_DIS
LIN {X 59.361,Y 89.031,Z 69.000,A 180.000,B 0.000,C 180.000} C_DIS
LIN {X 59.355,Y 89.030,Z 69.000,A 180.000,B 0.000,C 180.000} C_DIS
LIN {X 59.176,Y 89.020,Z 69.000,A 180.000,B 0.000,C 180.000} C_DIS
LIN {X 58.640,Y 89.003,Z 69.000,A 180.000,B 0.000,C 180.000} C_DIS
LIN {X 58.461,Y 89.000,Z 69.000,A 180.000,B 0.000,C 180.000} C_DIS
LIN {X 58.282,Y 89.006,Z 69.000,A 180.000,B 0.000,C 180.000} C_DIS
LIN {X 57.925,Y 89.017,Z 69.000,A 180.000,B 0.000,C 180.000} C_DIS
LIN {X 57.746,Y 89.023,Z 69.000,A 180.000,B 0.000,C 180.000} C_DIS
LIN {X 57.639,Y 89.031,Z 69.000,A 180.000,B 0.000,C 180.000} C_DIS
LIN {X 57.031,Y 89.088,Z 69.000,A 180.000,B 0.000,C 180.000} C_DIS
LIN {X 56.852,Y 89.110,Z 69.000,A 180.000,B 0.000,C 180.000} C_DIS
LIN {X 56.316,Y 89.195,Z 69.000,A 180.000,B 0.000,C 180.000} C_DIS
LIN {X 56.226,Y 89.209,Z 69.000,A 180.000,B 0.000,C 180.000} C_DIS
LIN {X 56.137,Y 89.225,Z 69.000,A 180.000,B 0.000,C 180.000} C_DIS
LIN {X 55.958,Y 89.265,Z 69.000,A 180.000,B 0.000,C 180.000} C_DIS
LIN {X 55.601,Y 89.345,Z 69.000,A 180.000,B 0.000,C 180.000} C_DIS
LIN {X 55.422,Y 89.385,Z 69.000,A 180.000,B 0.000,C 180.000} C_DIS
LIN {X 55.409,Y 89.388,Z 69.000,A 180.000,B 0.000,C 180.000} C_DIS
LIN {X 55.243,Y 89.434,Z 69.000,A 180.000,B 0.000,C 180.000} C_DIS
LIN {X 54.787,Y 89.567,Z 69.000,A 180.000,B 0.000,C 180.000} C_DIS
LIN {X 54.707,Y 89.590,Z 69.000,A 180.000,B 0.000,C 180.000} C_DIS
LIN {X 54.528,Y 89.650,Z 69.000,A 180.000,B 0.000,C 180.000} C_DIS
LIN {X 53.992,Y 89.843,Z 69.000,A 180.000,B 0.000,C 180.000} C_DIS
LIN {X 53.813,Y 89.913,Z 69.000,A 180.000,B 0.000,C 180.000} C_DIS
LIN {X 53.277,Y 90.146,Z 69.000,A 180.000,B 0.000,C 180.000} C_DIS
LIN {X 53.098,Y 90.229,Z 69.000,A 180.000,B 0.000,C 180.000} C_DIS
LIN {X 52.562,Y 90.502,Z 69.000,A 180.000,B 0.000,C 180.000} C_DIS
LIN {X 52.383,Y 90.601,Z 69.000,A 180.000,B 0.000,C 180.000} C_DIS
LIN {X 52.015,Y 90.818,Z 69.000,A 180.000,B 0.000,C 180.000} C_DIS
LIN {X 51.847,Y 90.918,Z 69.000,A 180.000,B 0.000,C 180.000} C_DIS
LIN {X 51.725,Y 90.997,Z 69.000,A 180.000,B 0.000,C 180.000} C_DIS
LIN {X 51.310,Y 91.279,Z 69.000,A 180.000,B 0.000,C 180.000} C_DIS
LIN {X 51.199,Y 91.355,Z 69.000,A 180.000,B 0.000,C 180.000} C_DIS
LIN {X 51.131,Y 91.403,Z 69.000,A 180.000,B 0.000,C 180.000} C_DIS
LIN {X 50.962,Y 91.533,Z 69.000,A 180.000,B 0.000,C 180.000} C_DIS
LIN {X 50.595,Y 91.818,Z 69.000,A 180.000,B 0.000,C 180.000} C_DIS
LIN {X 50.506,Y 91.891,Z 69.000,A 180.000,B 0.000,C 180.000} C_DIS
LIN {X 50.416,Y 91.969,Z 69.000,A 180.000,B 0.000,C 180.000} C_DIS
LIN {X 50.059,Y 92.284,Z 69.000,A 180.000,B 0.000,C 180.000} C_DIS
LIN {X 49.902,Y 92.427,Z 69.000,A 180.000,B 0.000,C 180.000} C_DIS
LIN {X 49.880,Y 92.449,Z 69.000,A 180.000,B 0.000,C 180.000} C_DIS
LIN {X 49.523,Y 92.807,Z 69.000,A 180.000,B 0.000,C 180.000} C_DIS
LIN {X 49.369,Y 92.964,Z 69.000,A 180.000,B 0.000,C 180.000} C_DIS
LIN {X 49.344,Y 92.991,Z 69.000,A 180.000,B 0.000,C 180.000} C_DIS
LIN {X 49.211,Y 93.142,Z 69.000,A 180.000,B 0.000,C 180.000} C_DIS
LIN {X 48.986,Y 93.397,Z 69.000,A 180.000,B 0.000,C 180.000} C_DIS
LIN {X 48.896,Y 93.500,Z 69.000,A 180.000,B 0.000,C 180.000} C_DIS
LIN {X 48.807,Y 93.609,Z 69.000,A 180.000,B 0.000,C 180.000} C_DIS
LIN {X 48.450,Y 94.070,Z 69.000,A 180.000,B 0.000,C 180.000} C_DIS
LIN {X 48.343,Y 94.215,Z 69.000,A 180.000,B 0.000,C 180.000} C_DIS
LIN {X 48.092,Y 94.584,Z 69.000,A 180.000,B 0.000,C 180.000} C_DIS
LIN {X 47.979,Y 94.751,Z 69.000,A 180.000,B 0.000,C 180.000} C_DIS
LIN {X 47.914,Y 94.855,Z 69.000,A 180.000,B 0.000,C 180.000} C_DIS
LIN {X 47.869,Y 94.930,Z 69.000,A 180.000,B 0.000,C 180.000} C_DIS
LIN {X 47.657,Y 95.288,Z 69.000,A 180.000,B 0.000,C 180.000} C_DIS
LIN {X 47.556,Y 95.460,Z 69.000,A 180.000,B 0.000,C 180.000} C_DIS
LIN {X 47.553,Y 95.466,Z 69.000,A 180.000,B 0.000,C 180.000} C_DIS
LIN {X 47.460,Y 95.645,Z 69.000,A 180.000,B 0.000,C 180.000} C_DIS
LIN {X 47.277,Y 96.003,Z 69.000,A 180.000,B 0.000,C 180.000} C_DIS
LIN {X 47.198,Y 96.159,Z 69.000,A 180.000,B 0.000,C 180.000} C_DIS
LIN {X 47.188,Y 96.181,Z 69.000,A 180.000,B 0.000,C 180.000} C_DIS
LIN {X 47.109,Y 96.360,Z 69.000,A 180.000,B 0.000,C 180.000} C_DIS
LIN {X 46.955,Y 96.718,Z 69.000,A 180.000,B 0.000,C 180.000} C_DIS
LIN {X 46.879,Y 96.897,Z 69.000,A 180.000,B 0.000,C 180.000} C_DIS
LIN {X 46.841,Y 96.997,Z 69.000,A 180.000,B 0.000,C 180.000} C_DIS
LIN {X 46.662,Y 97.494,Z 69.000,A 180.000,B 0.000,C 180.000} C_DIS
LIN {X 46.620,Y 97.612,Z 69.000,A 180.000,B 0.000,C 180.000} C_DIS
LIN {X 46.566,Y 97.790,Z 69.000,A 180.000,B 0.000,C 180.000} C_DIS
LIN {X 46.462,Y 98.148,Z 69.000,A 180.000,B 0.000,C 180.000} C_DIS
LIN {X 46.410,Y 98.327,Z 69.000,A 180.000,B 0.000,C 180.000} C_DIS
LIN {X 46.366,Y 98.505,Z 69.000,A 180.000,B 0.000,C 180.000} C_DIS
LIN {X 46.246,Y 99.042,Z 69.000,A 180.000,B 0.000,C 180.000} C_DIS
LIN {X 46.210,Y 99.221,Z 69.000,A 180.000,B 0.000,C 180.000} C_DIS
LIN {X 46.182,Y 99.399,Z 69.000,A 180.000,B 0.000,C 180.000} C_DIS
LIN {X 46.126,Y 99.753,Z 69.000,A 180.000,B 0.000,C 180.000} C_DIS
LIN {X 46.125,Y 99.757,Z 69.000,A 180.000,B 0.000,C 180.000} C_DIS
LIN {X 46.098,Y 99.936,Z 69.000,A 180.000,B 0.000,C 180.000} C_DIS
LIN {X 46.080,Y 100.114,Z 69.000,A 180.000,B 0.000,C 180.000} C_DIS
LIN {X 46.046,Y 100.472,Z 69.000,A 180.000,B 0.000,C 180.000} C_DIS
LIN {X 46.030,Y 100.651,Z 69.000,A 180.000,B 0.000,C 180.000} C_DIS
LIN {X 46.020,Y 100.829,Z 69.000,A 180.000,B 0.000,C 180.000} C_DIS
LIN {X 46.003,Y 101.366,Z 69.000,A 180.000,B 0.000,C 180.000} C_DIS
LIN {X 46.000,Y 101.545,Z 69.000,A 180.000,B 0.000,C 180.000} C_DIS
LIN {X 46.006,Y 101.723,Z 69.000,A 180.000,B 0.000,C 180.000} C_DIS
LIN {X 46.017,Y 102.081,Z 69.000,A 180.000,B 0.000,C 180.000} C_DIS
LIN {X 46.023,Y 102.260,Z 69.000,A 180.000,B 0.000,C 180.000} C_DIS
LIN {X 46.038,Y 102.438,Z 69.000,A 180.000,B 0.000,C 180.000} C_DIS
LIN {X 46.089,Y 102.975,Z 69.000,A 180.000,B 0.000,C 180.000} C_DIS
LIN {X 46.111,Y 103.153,Z 69.000,A 180.000,B 0.000,C 180.000} C_DIS
LIN {X 46.196,Y 103.690,Z 69.000,A 180.000,B 0.000,C 180.000} C_DIS
LIN {X 46.227,Y 103.869,Z 69.000,A 180.000,B 0.000,C 180.000} C_DIS
LIN {X 46.266,Y 104.047,Z 69.000,A 180.000,B 0.000,C 180.000} C_DIS
LIN {X 46.346,Y 104.405,Z 69.000,A 180.000,B 0.000,C 180.000} C_DIS
LIN {X 46.360,Y 104.467,Z 69.000,A 180.000,B 0.000,C 180.000} C_DIS
; Link Move Starts
LIN {X 46.439,Y 104.771,Z 69.000,A 180.000,B 0.000,C 180.000} C_DIS
LIN {X 46.527,Y 105.074,Z 68.999,A 180.000,B 0.000,C 180.000} C_DIS
LIN {X 46.616,Y 105.376,Z 68.998,A 180.000,B 0.000,C 180.000} C_DIS
LIN {X 46.722,Y 105.673,Z 68.996,A 180.000,B 0.000,C 180.000} C_DIS
LIN {X 46.829,Y 105.969,Z 68.994,A 180.000,B 0.000,C 180.000} C_DIS
LIN {X 46.946,Y 106.261,Z 68.991,A 180.000,B 0.000,C 180.000} C_DIS
LIN {X 47.071,Y 106.550,Z 68.988,A 180.000,B 0.000,C 180.000} C_DIS
LIN {X 47.198,Y 106.839,Z 68.985,A 180.000,B 0.000,C 180.000} C_DIS
LIN {X 47.340,Y 107.120,Z 68.981,A 180.000,B 0.000,C 180.000} C_DIS
LIN {X 47.483,Y 107.400,Z 68.977,A 180.000,B 0.000,C 180.000} C_DIS
LIN {X 47.636,Y 107.676,Z 68.972,A 180.000,B 0.000,C 180.000} C_DIS
LIN {X 47.716,Y 107.811,Z 68.969,A 180.000,B 0.000,C 180.000} C_DIS
LIN {X 47.796,Y 107.947,Z 68.967,A 180.000,B 0.000,C 180.000} C_DIS
LIN {X 47.876,Y 108.083,Z 68.964,A 180.000,B 0.000,C 180.000} C_DIS
LIN {X 47.958,Y 108.217,Z 68.961,A 180.000,B 0.000,C 180.000} C_DIS
LIN {X 48.046,Y 108.348,Z 68.959,A 180.000,B 0.000,C 180.000} C_DIS
LIN {X 48.135,Y 108.478,Z 68.956,A 180.000,B 0.000,C 180.000} C_DIS
LIN {X 48.223,Y 108.608,Z 68.952,A 180.000,B 0.000,C 180.000} C_DIS
LIN {X 48.312,Y 108.738,Z 68.949,A 180.000,B 0.000,C 180.000} C_DIS
LIN {X 48.402,Y 108.867,Z 68.946,A 180.000,B 0.000,C 180.000} C_DIS
LIN {X 48.498,Y 108.992,Z 68.943,A 180.000,B 0.000,C 180.000} C_DIS
LIN {X 48.595,Y 109.117,Z 68.939,A 180.000,B 0.000,C 180.000} C_DIS
LIN {X 48.691,Y 109.241,Z 68.936,A 180.000,B 0.000,C 180.000} C_DIS
LIN {X 48.788,Y 109.366,Z 68.932,A 180.000,B 0.000,C 180.000} C_DIS
LIN {X 48.886,Y 109.489,Z 68.928,A 180.000,B 0.000,C 180.000} C_DIS
LIN {X 48.990,Y 109.607,Z 68.925,A 180.000,B 0.000,C 180.000} C_DIS
LIN {X 49.094,Y 109.725,Z 68.921,A 180.000,B 0.000,C 180.000} C_DIS
LIN {X 49.198,Y 109.843,Z 68.917,A 180.000,B 0.000,C 180.000} C_DIS
LIN {X 49.302,Y 109.962,Z 68.913,A 180.000,B 0.000,C 180.000} C_DIS
LIN {X 49.408,Y 110.078,Z 68.909,A 180.000,B 0.000,C 180.000} C_DIS
LIN {X 49.519,Y 110.190,Z 68.905,A 180.000,B 0.000,C 180.000} C_DIS
LIN {X 49.631,Y 110.301,Z 68.900,A 180.000,B 0.000,C 180.000} C_DIS
LIN {X 49.742,Y 110.413,Z 68.896,A 180.000,B 0.000,C 180.000} C_DIS
LIN {X 49.853,Y 110.524,Z 68.892,A 180.000,B 0.000,C 180.000} C_DIS
LIN {X 49.966,Y 110.634,Z 68.887,A 180.000,B 0.000,C 180.000} C_DIS
LIN {X 50.084,Y 110.738,Z 68.883,A 180.000,B 0.000,C 180.000} C_DIS
LIN {X 50.202,Y 110.842,Z 68.878,A 180.000,B 0.000,C 180.000} C_DIS
LIN {X 50.321,Y 110.946,Z 68.873,A 180.000,B 0.000,C 180.000} C_DIS
LIN {X 50.439,Y 111.051,Z 68.869,A 180.000,B 0.000,C 180.000} C_DIS
LIN {X 50.559,Y 111.153,Z 68.864,A 180.000,B 0.000,C 180.000} C_DIS
LIN {X 50.683,Y 111.250,Z 68.859,A 180.000,B 0.000,C 180.000} C_DIS
LIN {X 50.807,Y 111.346,Z 68.854,A 180.000,B 0.000,C 180.000} C_DIS
LIN {X 50.869,Y 111.395,Z 68.851,A 180.000,B 0.000,C 180.000} C_DIS
LIN {X 50.932,Y 111.443,Z 68.849,A 180.000,B 0.000,C 180.000} C_DIS
LIN {X 50.994,Y 111.491,Z 68.846,A 180.000,B 0.000,C 180.000} C_DIS
LIN {X 51.056,Y 111.539,Z 68.844,A 180.000,B 0.000,C 180.000} C_DIS
LIN {X 51.118,Y 111.587,Z 68.841,A 180.000,B 0.000,C 180.000} C_DIS
LIN {X 51.182,Y 111.634,Z 68.839,A 180.000,B 0.000,C 180.000} C_DIS
LIN {X 51.247,Y 111.678,Z 68.836,A 180.000,B 0.000,C 180.000} C_DIS
LIN {X 51.377,Y 111.767,Z 68.831,A 180.000,B 0.000,C 180.000} C_DIS
LIN {X 51.508,Y 111.855,Z 68.825,A 180.000,B 0.000,C 180.000} C_DIS
LIN {X 51.638,Y 111.944,Z 68.820,A 180.000,B 0.000,C 180.000} C_DIS
LIN {X 51.703,Y 111.988,Z 68.817,A 180.000,B 0.000,C 180.000} C_DIS
LIN {X 51.768,Y 112.032,Z 68.815,A 180.000,B 0.000,C 180.000} C_DIS
LIN {X 51.835,Y 112.074,Z 68.812,A 180.000,B 0.000,C 180.000} C_DIS
LIN {X 51.902,Y 112.115,Z 68.809,A 180.000,B 0.000,C 180.000} C_DIS
LIN {X 51.970,Y 112.155,Z 68.807,A 180.000,B 0.000,C 180.000} C_DIS
LIN {X 52.106,Y 112.235,Z 68.801,A 180.000,B 0.000,C 180.000} C_DIS
LIN {X 52.309,Y 112.355,Z 68.793,A 180.000,B 0.000,C 180.000} C_DIS
LIN {X 52.377,Y 112.395,Z 68.790,A 180.000,B 0.000,C 180.000} C_DIS
LIN {X 52.445,Y 112.435,Z 68.787,A 180.000,B 0.000,C 180.000} C_DIS
LIN {X 52.514,Y 112.473,Z 68.785,A 180.000,B 0.000,C 180.000} C_DIS
LIN {X 52.584,Y 112.509,Z 68.782,A 180.000,B 0.000,C 180.000} C_DIS
LIN {X 52.724,Y 112.581,Z 68.776,A 180.000,B 0.000,C 180.000} C_DIS
LIN {X 52.794,Y 112.616,Z 68.774,A 180.000,B 0.000,C 180.000} C_DIS
LIN {X 52.935,Y 112.688,Z 68.768,A 180.000,B 0.000,C 180.000} C_DIS
LIN {X 53.075,Y 112.759,Z 68.763,A 180.000,B 0.000,C 180.000} C_DIS
LIN {X 53.145,Y 112.795,Z 68.760,A 180.000,B 0.000,C 180.000} C_DIS
LIN {X 53.217,Y 112.828,Z 68.757,A 180.000,B 0.000,C 180.000} C_DIS
LIN {X 53.289,Y 112.860,Z 68.754,A 180.000,B 0.000,C 180.000} C_DIS
LIN {X 53.361,Y 112.891,Z 68.752,A 180.000,B 0.000,C 180.000} C_DIS
LIN {X 53.506,Y 112.954,Z 68.746,A 180.000,B 0.000,C 180.000} C_DIS
LIN {X 53.723,Y 113.047,Z 68.738,A 180.000,B 0.000,C 180.000} C_DIS
LIN {X 53.795,Y 113.079,Z 68.735,A 180.000,B 0.000,C 180.000} C_DIS
LIN {X 53.867,Y 113.110,Z 68.732,A 180.000,B 0.000,C 180.000} C_DIS
LIN {X 53.941,Y 113.138,Z 68.730,A 180.000,B 0.000,C 180.000} C_DIS
LIN {X 54.015,Y 113.165,Z 68.727,A 180.000,B 0.000,C 180.000} C_DIS
LIN {X 54.163,Y 113.219,Z 68.721,A 180.000,B 0.000,C 180.000} C_DIS
LIN {X 54.237,Y 113.245,Z 68.719,A 180.000,B 0.000,C 180.000} C_DIS
LIN {X 54.385,Y 113.299,Z 68.713,A 180.000,B 0.000,C 180.000} C_DIS
LIN {X 54.533,Y 113.352,Z 68.708,A 180.000,B 0.000,C 180.000} C_DIS
LIN {X 54.607,Y 113.378,Z 68.705,A 180.000,B 0.000,C 180.000} C_DIS
LIN {X 54.682,Y 113.402,Z 68.702,A 180.000,B 0.000,C 180.000} C_DIS
LIN {X 54.758,Y 113.425,Z 68.699,A 180.000,B 0.000,C 180.000} C_DIS
LIN {X 54.834,Y 113.447,Z 68.697,A 180.000,B 0.000,C 180.000} C_DIS
LIN {X 54.985,Y 113.490,Z 68.691,A 180.000,B 0.000,C 180.000} C_DIS
LIN {X 55.287,Y 113.578,Z 68.680,A 180.000,B 0.000,C 180.000} C_DIS
LIN {X 55.363,Y 113.600,Z 68.677,A 180.000,B 0.000,C 180.000} C_DIS
LIN {X 55.440,Y 113.619,Z 68.675,A 180.000,B 0.000,C 180.000} C_DIS
LIN {X 55.516,Y 113.636,Z 68.672,A 180.000,B 0.000,C 180.000} C_DIS
LIN {X 55.670,Y 113.671,Z 68.666,A 180.000,B 0.000,C 180.000} C_DIS
LIN {X 55.824,Y 113.705,Z 68.661,A 180.000,B 0.000,C 180.000} C_DIS
LIN {X 56.054,Y 113.757,Z 68.653,A 180.000,B 0.000,C 180.000} C_DIS
LIN {X 56.131,Y 113.773,Z 68.650,A 180.000,B 0.000,C 180.000} C_DIS
LIN {X 56.209,Y 113.788,Z 68.647,A 180.000,B 0.000,C 180.000} C_DIS
LIN {X 56.286,Y 113.800,Z 68.644,A 180.000,B 0.000,C 180.000} C_DIS
LIN {X 56.442,Y 113.825,Z 68.639,A 180.000,B 0.000,C 180.000} C_DIS
LIN {X 56.831,Y 113.886,Z 68.625,A 180.000,B 0.000,C 180.000} C_DIS
LIN {X 56.909,Y 113.898,Z 68.622,A 180.000,B 0.000,C 180.000} C_DIS
LIN {X 56.987,Y 113.908,Z 68.620,A 180.000,B 0.000,C 180.000} C_DIS
LIN {X 57.065,Y 113.915,Z 68.617,A 180.000,B 0.000,C 180.000} C_DIS
LIN {X 57.536,Y 113.960,Z 68.600,A 180.000,B 0.000,C 180.000} C_DIS
LIN {X 57.614,Y 113.967,Z 68.598,A 180.000,B 0.000,C 180.000} C_DIS
LIN {X 57.693,Y 113.974,Z 68.595,A 180.000,B 0.000,C 180.000} C_DIS
LIN {X 57.771,Y 113.978,Z 68.592,A 180.000,B 0.000,C 180.000} C_DIS
LIN {X 57.850,Y 113.981,Z 68.589,A 180.000,B 0.000,C 180.000} C_DIS
LIN {X 58.244,Y 113.993,Z 68.576,A 180.000,B 0.000,C 180.000} C_DIS
LIN {X 58.401,Y 113.998,Z 68.570,A 180.000,B 0.000,C 180.000} C_DIS
LIN {X 58.480,Y 114.000,Z 68.567,A 180.000,B 0.000,C 180.000} C_DIS
LIN {X 58.558,Y 113.999,Z 68.565,A 180.000,B 0.000,C 180.000} C_DIS
LIN {X 58.637,Y 113.997,Z 68.562,A 180.000,B 0.000,C 180.000} C_DIS
LIN {X 59.188,Y 113.980,Z 68.543,A 180.000,B 0.000,C 180.000} C_DIS
LIN {X 59.267,Y 113.976,Z 68.540,A 180.000,B 0.000,C 180.000} C_DIS
LIN {X 59.345,Y 113.971,Z 68.537,A 180.000,B 0.000,C 180.000} C_DIS
LIN {X 59.424,Y 113.963,Z 68.534,A 180.000,B 0.000,C 180.000} C_DIS
LIN {X 59.973,Y 113.912,Z 68.515,A 180.000,B 0.000,C 180.000} C_DIS
LIN {X 60.051,Y 113.903,Z 68.512,A 180.000,B 0.000,C 180.000} C_DIS
LIN {X 60.129,Y 113.893,Z 68.510,A 180.000,B 0.000,C 180.000} C_DIS
LIN {X 60.207,Y 113.880,Z 68.507,A 180.000,B 0.000,C 180.000} C_DIS
LIN {X 60.751,Y 113.794,Z 68.488,A 180.000,B 0.000,C 180.000} C_DIS
LIN {X 60.829,Y 113.781,Z 68.485,A 180.000,B 0.000,C 180.000} C_DIS
LIN {X 60.906,Y 113.766,Z 68.482,A 180.000,B 0.000,C 180.000} C_DIS
LIN {X 60.983,Y 113.748,Z 68.479,A 180.000,B 0.000,C 180.000} C_DIS
LIN {X 61.521,Y 113.628,Z 68.460,A 180.000,B 0.000,C 180.000} C_DIS
LIN {X 61.598,Y 113.610,Z 68.457,A 180.000,B 0.000,C 180.000} C_DIS
LIN {X 61.674,Y 113.590,Z 68.455,A 180.000,B 0.000,C 180.000} C_DIS
LIN {X 61.749,Y 113.568,Z 68.452,A 180.000,B 0.000,C 180.000} C_DIS
LIN {X 62.279,Y 113.414,Z 68.433,A 180.000,B 0.000,C 180.000} C_DIS
LIN {X 62.354,Y 113.391,Z 68.430,A 180.000,B 0.000,C 180.000} C_DIS
LIN {X 62.429,Y 113.366,Z 68.427,A 180.000,B 0.000,C 180.000} C_DIS
LIN {X 62.503,Y 113.339,Z 68.424,A 180.000,B 0.000,C 180.000} C_DIS
LIN {X 62.873,Y 113.206,Z 68.411,A 180.000,B 0.000,C 180.000} C_DIS
LIN {X 63.021,Y 113.152,Z 68.405,A 180.000,B 0.000,C 180.000} C_DIS
LIN {X 63.095,Y 113.125,Z 68.402,A 180.000,B 0.000,C 180.000} C_DIS
LIN {X 63.168,Y 113.095,Z 68.400,A 180.000,B 0.000,C 180.000} C_DIS
LIN {X 63.313,Y 113.032,Z 68.394,A 180.000,B 0.000,C 180.000} C_DIS
LIN {X 63.746,Y 112.845,Z 68.378,A 180.000,B 0.000,C 180.000} C_DIS
LIN {X 63.818,Y 112.812,Z 68.375,A 180.000,B 0.000,C 180.000} C_DIS
LIN {X 63.889,Y 112.778,Z 68.372,A 180.000,B 0.000,C 180.000} C_DIS
LIN {X 64.169,Y 112.635,Z 68.361,A 180.000,B 0.000,C 180.000} C_DIS
LIN {X 64.450,Y 112.492,Z 68.350,A 180.000,B 0.000,C 180.000} C_DIS
LIN {X 64.520,Y 112.455,Z 68.347,A 180.000,B 0.000,C 180.000} C_DIS
LIN {X 64.588,Y 112.416,Z 68.345,A 180.000,B 0.000,C 180.000} C_DIS
LIN {X 64.792,Y 112.296,Z 68.336,A 180.000,B 0.000,C 180.000} C_DIS
LIN {X 64.859,Y 112.256,Z 68.334,A 180.000,B 0.000,C 180.000} C_DIS
LIN {X 64.995,Y 112.176,Z 68.328,A 180.000,B 0.000,C 180.000} C_DIS
LIN {X 65.130,Y 112.095,Z 68.323,A 180.000,B 0.000,C 180.000} C_DIS
LIN {X 65.198,Y 112.054,Z 68.320,A 180.000,B 0.000,C 180.000} C_DIS
LIN {X 65.263,Y 112.011,Z 68.317,A 180.000,B 0.000,C 180.000} C_DIS
LIN {X 65.654,Y 111.745,Z 68.301,A 180.000,B 0.000,C 180.000} C_DIS
LIN {X 65.785,Y 111.657,Z 68.295,A 180.000,B 0.000,C 180.000} C_DIS
LIN {X 65.849,Y 111.612,Z 68.292,A 180.000,B 0.000,C 180.000} C_DIS
LIN {X 65.912,Y 111.564,Z 68.290,A 180.000,B 0.000,C 180.000} C_DIS
LIN {X 66.036,Y 111.468,Z 68.284,A 180.000,B 0.000,C 180.000} C_DIS
LIN {X 66.223,Y 111.323,Z 68.276,A 180.000,B 0.000,C 180.000} C_DIS
LIN {X 66.347,Y 111.226,Z 68.270,A 180.000,B 0.000,C 180.000} C_DIS
LIN {X 66.410,Y 111.178,Z 68.268,A 180.000,B 0.000,C 180.000} C_DIS
LIN {X 66.471,Y 111.129,Z 68.265,A 180.000,B 0.000,C 180.000} C_DIS
LIN {X 66.531,Y 111.077,Z 68.262,A 180.000,B 0.000,C 180.000} C_DIS
LIN {X 66.708,Y 110.921,Z 68.254,A 180.000,B 0.000,C 180.000} C_DIS
LIN {X 66.826,Y 110.817,Z 68.248,A 180.000,B 0.000,C 180.000} C_DIS
LIN {X 66.885,Y 110.765,Z 68.246,A 180.000,B 0.000,C 180.000} C_DIS
LIN {X 67.003,Y 110.661,Z 68.240,A 180.000,B 0.000,C 180.000} C_DIS
LIN {X 67.062,Y 110.608,Z 68.237,A 180.000,B 0.000,C 180.000} C_DIS
LIN {X 67.118,Y 110.553,Z 68.235,A 180.000,B 0.000,C 180.000} C_DIS
LIN {X 67.229,Y 110.441,Z 68.229,A 180.000,B 0.000,C 180.000} C_DIS
LIN {X 67.396,Y 110.274,Z 68.221,A 180.000,B 0.000,C 180.000} C_DIS
LIN {X 67.508,Y 110.163,Z 68.215,A 180.000,B 0.000,C 180.000} C_DIS
LIN {X 67.563,Y 110.107,Z 68.213,A 180.000,B 0.000,C 180.000} C_DIS
LIN {X 67.618,Y 110.051,Z 68.210,A 180.000,B 0.000,C 180.000} C_DIS
LIN {X 67.671,Y 109.992,Z 68.207,A 180.000,B 0.000,C 180.000} C_DIS
LIN {X 67.827,Y 109.815,Z 68.199,A 180.000,B 0.000,C 180.000} C_DIS
LIN {X 67.931,Y 109.697,Z 68.193,A 180.000,B 0.000,C 180.000} C_DIS
LIN {X 68.035,Y 109.579,Z 68.188,A 180.000,B 0.000,C 180.000} C_DIS
LIN {X 68.087,Y 109.520,Z 68.185,A 180.000,B 0.000,C 180.000} C_DIS
LIN {X 68.138,Y 109.459,Z 68.182,A 180.000,B 0.000,C 180.000} C_DIS
LIN {X 68.187,Y 109.398,Z 68.180,A 180.000,B 0.000,C 180.000} C_DIS
LIN {X 68.284,Y 109.273,Z 68.174,A 180.000,B 0.000,C 180.000} C_DIS
LIN {X 68.380,Y 109.149,Z 68.169,A 180.000,B 0.000,C 180.000} C_DIS
LIN {X 68.477,Y 109.024,Z 68.164,A 180.000,B 0.000,C 180.000} C_DIS
LIN {X 68.525,Y 108.962,Z 68.161,A 180.000,B 0.000,C 180.000} C_DIS
LIN {X 68.573,Y 108.900,Z 68.159,A 180.000,B 0.000,C 180.000} C_DIS
LIN {X 68.620,Y 108.837,Z 68.156,A 180.000,B 0.000,C 180.000} C_DIS
LIN {X 68.665,Y 108.772,Z 68.154,A 180.000,B 0.000,C 180.000} C_DIS
LIN {X 68.710,Y 108.707,Z 68.151,A 180.000,B 0.000,C 180.000} C_DIS
LIN {X 68.754,Y 108.642,Z 68.149,A 180.000,B 0.000,C 180.000} C_DIS
LIN {X 68.842,Y 108.512,Z 68.144,A 180.000,B 0.000,C 180.000} C_DIS
LIN {X 68.931,Y 108.381,Z 68.139,A 180.000,B 0.000,C 180.000} C_DIS
LIN {X 69.019,Y 108.251,Z 68.134,A 180.000,B 0.000,C 180.000} C_DIS
LIN {X 69.103,Y 108.118,Z 68.129,A 180.000,B 0.000,C 180.000} C_DIS
LIN {X 69.183,Y 107.982,Z 68.124,A 180.000,B 0.000,C 180.000} C_DIS
LIN {X 69.263,Y 107.846,Z 68.120,A 180.000,B 0.000,C 180.000} C_DIS
LIN {X 69.344,Y 107.711,Z 68.115,A 180.000,B 0.000,C 180.000} C_DIS
LIN {X 69.424,Y 107.575,Z 68.111,A 180.000,B 0.000,C 180.000} C_DIS
LIN {X 69.499,Y 107.437,Z 68.106,A 180.000,B 0.000,C 180.000} C_DIS
LIN {X 69.570,Y 107.296,Z 68.102,A 180.000,B 0.000,C 180.000} C_DIS
LIN {X 69.642,Y 107.156,Z 68.097,A 180.000,B 0.000,C 180.000} C_DIS
LIN {X 69.713,Y 107.016,Z 68.093,A 180.000,B 0.000,C 180.000} C_DIS
LIN {X 69.785,Y 106.875,Z 68.089,A 180.000,B 0.000,C 180.000} C_DIS
LIN {X 69.851,Y 106.732,Z 68.085,A 180.000,B 0.000,C 180.000} C_DIS
LIN {X 69.913,Y 106.588,Z 68.081,A 180.000,B 0.000,C 180.000} C_DIS
LIN {X 69.976,Y 106.443,Z 68.077,A 180.000,B 0.000,C 180.000} C_DIS
LIN {X 70.038,Y 106.299,Z 68.073,A 180.000,B 0.000,C 180.000} C_DIS
LIN {X 70.101,Y 106.154,Z 68.070,A 180.000,B 0.000,C 180.000} C_DIS
LIN {X 70.158,Y 106.007,Z 68.066,A 180.000,B 0.000,C 180.000} C_DIS
LIN {X 70.211,Y 105.859,Z 68.062,A 180.000,B 0.000,C 180.000} C_DIS
LIN {X 70.264,Y 105.711,Z 68.059,A 180.000,B 0.000,C 180.000} C_DIS
LIN {X 70.318,Y 105.563,Z 68.056,A 180.000,B 0.000,C 180.000} C_DIS
LIN {X 70.371,Y 105.414,Z 68.052,A 180.000,B 0.000,C 180.000} C_DIS
LIN {X 70.418,Y 105.264,Z 68.049,A 180.000,B 0.000,C 180.000} C_DIS
LIN {X 70.462,Y 105.113,Z 68.046,A 180.000,B 0.000,C 180.000} C_DIS
